(* CODESYS project Parostol_V4.2.project
   CompiledLibraryCompatibilityVersion: CODESYS V3.5 SP16 Patch 3

Project tree, tasks and I/O mapping:
  Device : PLC210, Production association OWEN, order no. 1, version 3.5.17.31
    application Application
      libraries: Standard, * (System); VisuDialogs, * (System); BASIC, 3.3.3.0 (OSCAT); Local Time Library, 3.5.3.50 (Andrew Sorokin); BUILDING, 1.0.0.0 (OSCAT); CmpOwenPidRegs, 3.5.14.33 (Production association OWEN); VisuElemsDateTime Interfaces, * (Intern); CmpBitmapPool, * (System); VisuElemXYChart, 4.1.0.0 (System); CAA DTUtil Extern, 3.5.17.0 (CAA Technical Workgroup); EtherCATStack, 4.2.0.0 (3S - Smart Software Solutions GmbH); Trace Mgr Utils, 4.1.0.0 (Intern); VisuFPlot, 4.1.0.0 (Intern); CmpTargetVisu, 3.5.17.0 (System); CAA Mathematics, 3.5.17.0 (CAA Technical Workgroup); OwenArchiverErrors, 3.5.4.3 (Production association OWEN); Standard64, * (System); OwenStringUtils, 3.5.4.8 (Production association OWEN); cmpSysExec, 3.5.11.30 (OWEN); StringUtils, 3.5.17.0 (System); Util, * (System); Mx210 Assistant, 3.5.11.5 (Production association OWEN)
      Parostol_Zadanie/
        task MainTask (cyclic, interval 20 ms, priority 1) calls PLC_PRG_Stol_1, PLC_PRG_Stol_2, PLC_PRG_Stol_3, PLC_PRG_Stol_4, PLC_PRG_CFC_Davlenie_Stol_1_2, PLC_PRG_CFC_Davlenie_Stol_3_4, PLC_PRG_CFC_Temperatura_Stol_1, PLC_PRG_CFC_Temperatura_Stol_3, PLC_PRG_CFC_Temperatura_Stol_4, PLC_PRG_archive, Connection
        task TrendRecordingTask (cyclic, interval 5000 ms, priority 31) calls VisuTrendStorageAccess.GlobalInstances.g_TrendRecordingManager.CyclicCall
        task VISU_TASK (cyclic, interval 40 ms, priority 0) calls VisuElems.Visu_Prg
        task OwenCloudTask (cyclic, interval 50 ms, priority 31) calls OwenStorage.CLOUD_PRG
        task DatasourcesTask (cyclic, interval 50 ms, priority 31) calls nothing
        task OwenArchiver (cyclic, interval T#100ms, priority 10) calls OwenArchiverDrivers.Archive_Prg
        program PLC_PRG_Stol_1 [CFC]
        function block GRAPH [ST]
        visualisation Zadanie_1
        visualisation HOME_1
        Trend Recording Manager
          Visualization_Trend_Stol_1
          Visualization_Trend_Stol_2
          TrendRecording_CFC_Davlenie_1_2
          TrendRecording_CFC_Temperatura_1
          Visualization_Trend_Stol_3
          Visualization_Trend_Stol_4
        visualisation Visualization_CFC_Davlenie_1_2
        visualisation HOME
        visualisation MnemoScheme
        visualisation Journal
        visualisation Zadanie_2
        program PLC_PRG_Stol_2 [CFC]
        visualisation Visualization_CFC_Temperatura_1
        program PLC_PRG_Stol_3 [CFC]
        program PLC_PRG_Stol_4 [CFC]
        visualisation Zadanie_3
        visualisation Zadanie_4
        visualisation Visualization_CFC_Temperatura_4
        visualisation Visualization_CFC_Temperatura_2
        visualisation Visualization_CFC_Temperatura_3
        visualisation Visualization_CFC_Davlenie_3_4
      CFC_Davlenie_PID/
        program PLC_PRG_CFC_Davlenie_Stol_1_2 [CFC]
        program PLC_PRG_CFC_Davlenie_Stol_3_4 [CFC]
      global variables GVL
      CFC_Temperatura_PID/
        function CheckPidParams_CFC [CFC]
        program PLC_PRG_CFC_Temperatura_Stol_1 [CFC]
        program PLC_PRG_CFC_Temperatura_Stol_4 [CFC]
        program PLC_PRG_CFC_Temperatura_Stol_3 [CFC]
        program PLC_PRG_CFC_Temperatura_Stol_2 [CFC]
      TargetVariables/
        global variables TargetVars
        data type TRG_LeftSide
        data type TRG_Debug
        data type TRG_Drives
        data type TRG_Info
        data type TRG_PLC210
        data type TRG_RTC
        data type TRG_Watchdog
        data type TRG_RightSide
        data type TRG_Buzzer
      global variables PID_GLOBALS
      Списки текстов/
        text list ANR_MODE
        text list ANR_WAVE_COUNT
        text list ERROR_PID
        text list STATE_PID
      archive/
        program PLC_PRG_archive [ST]: act01_DriveInfo
        data type DriveInfo
        function REAL_TO_FWSTRING [ST]
        function BYTE_SIZE_TO_WSTRING [ST]
      program Connection [ST]
      Symbols
      instructions/
        visualisation HELP
        visualisation zapros
        visualisation instrykcai_avtoriz
      global variables NVI_RETAIN
    Ethernet : Ethernet, 3S - Smart Software Solutions GmbH, version 3.5.17.0
        settings: IPAddress = [192,168,0,228]; SubnetMask = [255,255,255,0]; GatewayAddress = [0,0,0,0]; SaveCommunicationSettings = FALSE
      Modbus_TCP_Master : Modbus TCP Master, 3S - Smart Software Solutions GmbH, version 3.5.17.0
        MK210_311_Stol_1_2 : MK210-311, Production association OWEN, version 3.5.11.7
            settings: IPAddress = [192, 168, 0, 230]
            output Application.PLC_PRG_CFC_Davlenie_Stol_1_2.xMore : BOOL  // Битовая маска выходов (запись).Выход 1
            output Application.PLC_PRG_CFC_Davlenie_Stol_1_2.xLess : BOOL  // Битовая маска выходов (запись).Выход 2
            output Application.PLC_PRG_CFC_Temperatura_Stol_1.xLess : BOOL  // Битовая маска выходов (запись).Выход 3
            output Application.PLC_PRG_CFC_Temperatura_Stol_1.xMore : BOOL  // Битовая маска выходов (запись).Выход 4
            unmapped channels: Tmp, Исключить модуль из опроса, Флаг ошибки, Битовая маска входов, Битовая маска выходов (чтение), Битовая маска выходов (запись), Битовая маска диагностики выходов, Значение счетчика, Значение счетчика, Значение счетчика, Значение счетчика, Значение счетчика, Значение счетчика, Сбросить счетчик, Сбросить счетчик, Сбросить счетчик, Сбросить счетчик, Сбросить счетчик, Сбросить счетчик, Период ШИМ (чтение), Период ШИМ (чтение), Период ШИМ (чтение), Период ШИМ (чтение), Период ШИМ (чтение), Период ШИМ (чтение), Период ШИМ (чтение), Период ШИМ (чтение), Период ШИМ (запись), Период ШИМ (запись), Период ШИМ (запись), Период ШИМ (запись), Период ШИМ (запись), Период ШИМ (запись), Период ШИМ (запись), Период ШИМ (запись), Коэффициент заполнения ШИМ (чтение), Коэффициент заполнения ШИМ (чтение), Коэффициент заполнения ШИМ (чтение), Коэффициент заполнения ШИМ (чтение), Коэффициент заполнения ШИМ (чтение),
              Коэффициент заполнения ШИМ (чтение), Коэффициент заполнения ШИМ (чтение), Коэффициент заполнения ШИМ (чтение), Коэффициент заполнения ШИМ (запись), Коэффициент заполнения ШИМ (запись), Коэффициент заполнения ШИМ (запись), Коэффициент заполнения ШИМ (запись), Коэффициент заполнения ШИМ (запись), Коэффициент заполнения ШИМ (запись), Коэффициент заполнения ШИМ (запись), Коэффициент заполнения ШИМ (запись)
        MV210_212_Stol_1_2 : MV210-212, Production association OWEN, version 3.5.11.7
            settings: IPAddress = [192, 168, 0, 231]
            unmapped channels: Tmp, Исключить модуль из опроса, Флаг ошибки, Битовая маска входов, Значение, Значение, Значение, Значение, Значение, Значение, Значение, Значение, Значение счетчика, Значение счетчика, Значение счетчика, Значение счетчика, Значение счетчика, Значение счетчика, Значение счетчика, Значение счетчика, Значение счетчика, Значение счетчика, Значение счетчика, Значение счетчика, Значение счетчика, Значение счетчика, Значение счетчика, Значение счетчика, Значение счетчика, Значение счетчика, Значение счетчика, Значение счетчика, Значение счетчика, Значение счетчика, Значение счетчика, Значение счетчика, Сбросить значение, Сбросить значение, Сбросить значение, Сбросить значение,
              Сбросить значение, Сбросить значение, Сбросить значение, Сбросить значение, Сбросить счетчик, Сбросить счетчик, Сбросить счетчик, Сбросить счетчик, Сбросить счетчик, Сбросить счетчик, Сбросить счетчик, Сбросить счетчик, Сбросить счетчик, Сбросить счетчик, Сбросить счетчик, Сбросить счетчик, Сбросить счетчик, Сбросить счетчик, Сбросить счетчик, Сбросить счетчик, Сбросить счетчик, Сбросить счетчик, Сбросить счетчик, Сбросить счетчик, Сбросить счетчик, Сбросить счетчик, Сбросить счетчик, Сбросить счетчик
        MV210_101_Stol_1_2 : MV210-101, Production association OWEN, version 3.5.11.7
            settings: IPAddress = [192, 168, 0, 232]; Ииспользовать настройки конфигурации = FALSE
            input  Application.PID_GLOBALS.g_rCurrentValue_Temperatura_Stol_1 : REAL  // Вход 3.Значение
            input  Application.PID_GLOBALS.g_rCurrentValue_Davlenie_Podacha_Stol_1_2 : REAL  // Вход 5.Значение
            input  Application.PID_GLOBALS.g_wSampleTime_Davlenie_Stol_1_2 : UINT  // Вход 5.Циклическое время
            input  Application.PID_GLOBALS.g_rCurrentValue_Davlenie_Obratnaja_Stol_1_2 : REAL  // Вход 6.Значение
            unmapped channels: Tmp, Исключить модуль из опроса, Флаг ошибки, Записать настройки, Прочитать настройки, Вход 1 (чтение), Вход 2 (чтение), Вход 3 (чтение), Вход 4 (чтение), Вход 5 (чтение), Вход 6 (чтение), Вход 7 (чтение), Вход 8 (чтение), Вход 1 (запись), Вход 2 (запись), Вход 3 (запись), Вход 4 (запись), Вход 5 (запись), Вход 6 (запись), Вход 7 (запись), Вход 8 (запись), Вход 1, Вход 2, Вход 3, Вход 4, Вход 5, Вход 6, Вход 7, Вход 8
        MK210_311_Stol_3_4 : MK210-311, Production association OWEN, version 3.5.11.7
            settings: IPAddress = [192, 168, 0, 233]
            output Application.PLC_PRG_CFC_Davlenie_Stol_3_4.xMore : BOOL  // Битовая маска выходов (запись).Выход 1
            output Application.PLC_PRG_CFC_Davlenie_Stol_3_4.xLess : BOOL  // Битовая маска выходов (запись).Выход 2
            output Application.PLC_PRG_CFC_Temperatura_Stol_3.xMore : BOOL  // Битовая маска выходов (запись).Выход 3
            output Application.PLC_PRG_CFC_Temperatura_Stol_3.xLess : BOOL  // Битовая маска выходов (запись).Выход 4
            output Application.PLC_PRG_CFC_Temperatura_Stol_4.xMore : BOOL  // Битовая маска выходов (запись).Выход 5
            output Application.PLC_PRG_CFC_Temperatura_Stol_4.xLess : BOOL  // Битовая маска выходов (запись).Выход 6
            unmapped channels: Tmp, Исключить модуль из опроса, Флаг ошибки, Битовая маска входов, Битовая маска выходов (чтение), Битовая маска выходов (запись), Битовая маска диагностики выходов, Значение счетчика, Значение счетчика, Значение счетчика, Значение счетчика, Значение счетчика, Значение счетчика, Сбросить счетчик, Сбросить счетчик, Сбросить счетчик, Сбросить счетчик, Сбросить счетчик, Сбросить счетчик, Период ШИМ (чтение), Период ШИМ (чтение), Период ШИМ (чтение), Период ШИМ (чтение), Период ШИМ (чтение), Период ШИМ (чтение), Период ШИМ (чтение), Период ШИМ (чтение), Период ШИМ (запись), Период ШИМ (запись), Период ШИМ (запись), Период ШИМ (запись), Период ШИМ (запись), Период ШИМ (запись), Период ШИМ (запись), Период ШИМ (запись), Коэффициент заполнения ШИМ (чтение), Коэффициент заполнения ШИМ (чтение), Коэффициент заполнения ШИМ (чтение), Коэффициент заполнения ШИМ (чтение), Коэффициент заполнения ШИМ (чтение),
              Коэффициент заполнения ШИМ (чтение), Коэффициент заполнения ШИМ (чтение), Коэффициент заполнения ШИМ (чтение), Коэффициент заполнения ШИМ (запись), Коэффициент заполнения ШИМ (запись), Коэффициент заполнения ШИМ (запись), Коэффициент заполнения ШИМ (запись), Коэффициент заполнения ШИМ (запись), Коэффициент заполнения ШИМ (запись), Коэффициент заполнения ШИМ (запись), Коэффициент заполнения ШИМ (запись)
        MV210_212_Stol_3_4 : MV210-212, Production association OWEN, version 3.5.11.7
            settings: IPAddress = [192, 168, 0, 234]
            unmapped channels: Tmp, Исключить модуль из опроса, Флаг ошибки, Битовая маска входов, Значение, Значение, Значение, Значение, Значение, Значение, Значение, Значение, Значение счетчика, Значение счетчика, Значение счетчика, Значение счетчика, Значение счетчика, Значение счетчика, Значение счетчика, Значение счетчика, Значение счетчика, Значение счетчика, Значение счетчика, Значение счетчика, Значение счетчика, Значение счетчика, Значение счетчика, Значение счетчика, Значение счетчика, Значение счетчика, Значение счетчика, Значение счетчика, Значение счетчика, Значение счетчика, Значение счетчика, Значение счетчика, Сбросить значение, Сбросить значение, Сбросить значение, Сбросить значение,
              Сбросить значение, Сбросить значение, Сбросить значение, Сбросить значение, Сбросить счетчик, Сбросить счетчик, Сбросить счетчик, Сбросить счетчик, Сбросить счетчик, Сбросить счетчик, Сбросить счетчик, Сбросить счетчик, Сбросить счетчик, Сбросить счетчик, Сбросить счетчик, Сбросить счетчик, Сбросить счетчик, Сбросить счетчик, Сбросить счетчик, Сбросить счетчик, Сбросить счетчик, Сбросить счетчик, Сбросить счетчик, Сбросить счетчик, Сбросить счетчик, Сбросить счетчик, Сбросить счетчик, Сбросить счетчик
        MV210_101_Stol_3_4 : MV210-101, Production association OWEN, version 3.5.11.7
            settings: IPAddress = [192, 168, 0, 235]; Ииспользовать настройки конфигурации = FALSE
            input  Application.PID_GLOBALS.g_rCurrentValue_Temperatura_Stol_3 : REAL  // Вход 1.Значение
            input  Application.PID_GLOBALS.g_rCurrentValue_Temperatura_Stol_4 : REAL  // Вход 3.Значение
            input  Application.PID_GLOBALS.g_rCurrentValue_Davlenie_Podacha_Stol_3_4 : REAL  // Вход 5.Значение
            input  Application.PID_GLOBALS.g_wSampleTime_Davlenie_Stol_3_4 : UINT  // Вход 5.Циклическое время
            input  Application.PID_GLOBALS.g_rCurrentValue_Davlenie_Obratnaja_Stol_3_4 : REAL  // Вход 6.Значение
            unmapped channels: Tmp, Исключить модуль из опроса, Флаг ошибки, Записать настройки, Прочитать настройки, Вход 1 (чтение), Вход 2 (чтение), Вход 3 (чтение), Вход 4 (чтение), Вход 5 (чтение), Вход 6 (чтение), Вход 7 (чтение), Вход 8 (чтение), Вход 1 (запись), Вход 2 (запись), Вход 3 (запись), Вход 4 (запись), Вход 5 (запись), Вход 6 (запись), Вход 7 (запись), Вход 8 (запись), Вход 1, Вход 2, Вход 3, Вход 4, Вход 5, Вход 6, Вход 7, Вход 8
    PLC210_01 : PLC210-02, Production association OWEN, version 3.5.17.3001
        unmapped channels: Канал питания 1, Канал питания 2, Сервисная кнопка, Температура CPU, Переключатель Старт\Стоп
      LeftSide : LeftSide-01, Production association OWEN, version 3.5.17.3001
          unmapped channels: Битовая маска входов, Значение счетчика, Значение счетчика, Значение счетчика, Значение счетчика, Значение счетчика, Значение счетчика, Значение счетчика, Значение счетчика, Значение счетчика, Значение счетчика, Значение счетчика, Значение счетчика, Период импульса, Период импульса, Период импульса, Период импульса, Период импульса, Период импульса, Период импульса, Период импульса, Период импульса, Период импульса, Период импульса, Период импульса, Длительность импульса, Длительность импульса, Длительность импульса, Длительность импульса, Длительность импульса, Длительность импульса, Длительность импульса, Длительность импульса, Длительность импульса, Длительность импульса, Длительность импульса, Длительность импульса, Осталось сгенерировать импульсов, Осталось сгенерировать импульсов, Осталось сгенерировать импульсов,
            Осталось сгенерировать импульсов, Битовая маска диагностики выходов, Счётчик ошибок выхода 1, Счётчик ошибок выхода 2, Счётчик ошибок выхода 3, Счётчик ошибок выхода 4, Количество импульсов AB энкодера 1, Количество импульсов AB энкодера 2, Количество импульсов AB энкодера 3, Количество импульсов AB энкодера 4, Количество импульсов AB энкодера 5, Количество импульсов AB энкодера 6, Количество импульсов ABZ энкодера 1, Количество импульсов ABZ энкодера 2, Количество импульсов ABZ энкодера 3, Количество оборотов ABZ энкодера 1, Количество оборотов ABZ энкодера 2, Количество оборотов ABZ энкодера 3, Битовая маска выходов (запись), Количество импульсов генератора (запись), Количество импульсов генератора (запись), Количество импульсов генератора (запись), Количество импульсов генератора (запись), Выход 1, Выход 2, Выход 3, Выход 4
      RightSide : RightSide-02, Production association OWEN, version 3.5.17.3001
          unmapped channels: Наличие связи, Счетчик ошибок, Битовая маска входов, Битовая маска выходов (запись)
    OwenRTC : OwenRTC, Production association OWEN, version 3.5.17.3001
        input  Application.GVL.hour AT %IB268 : USINT  // Hour
        input  Application.GVL.minute : USINT  // Minute
        input  Application.GVL.day_of_week : USINT  // Day of Week
        unmapped channels: Year, Month, Day, Second, Week of Year, Format Date, Format Time, UTC Offset, NTP Enabled, NTP Error, System Timer, Date And Time, Operating Time, New Year, New Month, New Day, New Hour, New Minute, New Second, New UTC Offset, Set Settings DT, Enable NTP, Prefer Server
    OwenCloud : OwenCloud, Production association OWEN, version 3.5.17.3001
        unmapped channels: OwenCloud enabled, Folder error, Symbol error, No Symbol Config, Status, Enable OwenCloud
    Buzzer : Buzzer, Production association OWEN, version 3.5.17.3001
        unmapped channels: Buzzer enabled, Enable Buzzer, Sound frequency
    Drives : Drives, Production association OWEN, version 3.5.17.3001
        input  Application.PLC_PRG_archive.stPlcMemory.uleFullSize : ULINT  // FS size
        input  Application.PLC_PRG_archive.stPlcMemory.uleUsedSize : ULINT  // FS used
        input  Application.PLC_PRG_archive.stPlcMemory.uleFreeSize : ULINT  // FS free
        input  Application.PLC_PRG_archive.stUsbMemory.xIsMounted : BIT  // USB Mounted
        input  Application.PLC_PRG_archive.stUsbMemory.xUnmountDone : BIT  // USB Unmount done
        input  Application.PLC_PRG_archive.stUsbMemory.uleFullSize : ULINT  // USB size
        input  Application.PLC_PRG_archive.stUsbMemory.uleUsedSize : ULINT  // USB used
        input  Application.PLC_PRG_archive.stUsbMemory.uleFreeSize : ULINT  // USB free
        output Application.PID_GLOBALS.Start_USB_arv : BIT  // Enable Drives
        output Application.PLC_PRG_archive.stUsbMemory.xUnmount : BIT  // USB Unmount
        unmapped channels: MMC Mounted, MMC Unmount done, MMC size, MMC used, MMC free, FS wear, MMC Unmount
    Debug : Debug, Production association OWEN, version 3.5.17.3001
        unmapped channels: RAM used, RAM free, Open files, Processor usage, Core temp, Enable Debug, Debug pause
    Info : Info, Production association OWEN, version 3.5.17.3001
        unmapped channels: VENDOR, DEVICE, SERIAL, RUNTIME, FIRMWARE, LINUX, TARGET, PROJECT, AUTHOR, VERSION, PROFILE, LASTCHANGES
    Watchdog : Watchdog, Production association OWEN, version 3.5.17.3001
        unmapped channels: Exception Handling, Last Exception Code, Last Exception Description, Last Exception Time, Hardware Watchdog Flag, Power Reboot Count, Watchdog Reboot Count, Exception Reboot Count, Command Reboot Count, Reboot, Reset Counters
    OwenArchiver : OwenArchiver, Production association OWEN, version 3.5.4.9
        settings: Имя архива = 'STOL_1'
        output Application.PID_GLOBALS.xGO : BIT  // Запустить архиватор
        output Application.PID_GLOBALS.zGO : BIT  // Команда записи
        input  Application.PLC_PRG_archive.xArchError_1 : USINT  // Код последней ошибки
        input  Application.PLC_PRG_archive.xArchStatus_1 : BIT  // Архиватор работает
        unmapped channels: Запись лога отладки, Путь архивации, Имя архива, Использование буфера записи, Размер архива
      CSVFormat : CSVFormat, Production association OWEN, version 3.5.4.9
      REAL_Variable : REAL Variable, Production association OWEN, version 3.5.4.9
          settings: Описание переменной = 'Выставленное_давление'
          output Application.PLC_PRG_CFC_Davlenie_Stol_1_2.Davlenie_Stol_1_2_rSetPoint : REAL  // Переменная
      BYTE_Stol_1_MINUTE_PONEDEL : BYTE Variable, Production association OWEN, version 3.5.4.9
          settings: Описание переменной = 'Минуты_понедельник'
          output Application.NVI_RETAIN.minuteMondayStolOne : BYTE  // Переменная
      REAL_Stol_1_Y1 : REAL Variable, Production association OWEN, version 3.5.4.9
          settings: Описание переменной = 'Температура_стола'
          output Application.PLC_PRG_Stol_1.Y1 : REAL  // Переменная
      REAL_Stol_1_Y2 : REAL Variable, Production association OWEN, version 3.5.4.9
          settings: Описание переменной = 'Температура_подъема'
          output Application.PLC_PRG_Stol_1.Y2 : REAL  // Переменная
      REAL_Stol_1_Y3 : REAL Variable, Production association OWEN, version 3.5.4.9
          settings: Описание переменной = 'Температура_выдержки'
          output Application.PLC_PRG_Stol_1.Y3 : REAL  // Переменная
      REAL_Stoll_1_HX2 : REAL Variable, Production association OWEN, version 3.5.4.9
          settings: Описание переменной = 'Время_подъема_часы'
          output Application.PLC_PRG_Stol_1.HX2 : REAL  // Переменная
      REAL_Stol_1_MX2 : REAL Variable, Production association OWEN, version 3.5.4.9
          settings: Описание переменной = 'Время_подъема_минуты'
          output Application.PLC_PRG_Stol_1.MX2 : REAL  // Переменная
      REAL_Stol_1_HX3 : REAL Variable, Production association OWEN, version 3.5.4.9
          settings: Описание переменной = 'Время_выдержки_часы'
          output Application.PLC_PRG_Stol_1.HX3 : REAL  // Переменная
      REAL_Stol_1_MX3 : REAL Variable, Production association OWEN, version 3.5.4.9
          settings: Описание переменной = 'Время_выдержки_минуты'
          output Application.PLC_PRG_Stol_1.MX3 : REAL  // Переменная
      BYTE_Stol_1_HOUR_PONEDEL : BYTE Variable, Production association OWEN, version 3.5.4.9
          settings: Описание переменной = 'Час_понедельник'
          output Application.NVI_RETAIN.hourMondayStolOne : BYTE  // Переменная
      BYTE_Stol_1_HOUR_VTORN : BYTE Variable, Production association OWEN, version 3.5.4.9
          settings: Описание переменной = 'Час_вторник'
          output Application.NVI_RETAIN.hourTuesdayStolOne : BYTE  // Переменная
      BYTE_Stol_1_MINUTE_VTORN : BYTE Variable, Production association OWEN, version 3.5.4.9
          settings: Описание переменной = 'Минуты_вторник'
          output Application.NVI_RETAIN.minuteTuesdayStolOne : BYTE  // Переменная
      BYTE_Stol_1_HOUR_SREDA : BYTE Variable, Production association OWEN, version 3.5.4.9
          settings: Описание переменной = 'Час_среды'
          output Application.NVI_RETAIN.hourWednesdayStolOne : BYTE  // Переменная
      BYTE_Stol_1_MINUTE_SREDA : BYTE Variable, Production association OWEN, version 3.5.4.9
          settings: Описание переменной = 'Минуты_среды'
          output Application.NVI_RETAIN.minuteWednesdayStolOne : BYTE  // Переменная
      BYTE_Stol_1_PONEDEL_BYTE : BYTE Variable, Production association OWEN, version 3.5.4.9
          settings: Описание переменной = 'Флаг_понедельника'
          output Application.PLC_PRG_Stol_1.PONEDEL_BYTE : BYTE  // Переменная
      BYTE_Stol_1_VTORN_BYTE : BYTE Variable, Production association OWEN, version 3.5.4.9
          settings: Описание переменной = 'Флаг_вторника'
          output Application.PLC_PRG_Stol_1.VTORN_BYTE : BYTE  // Переменная
      BYTE_Stol_1_SREDA_BYTE : BYTE Variable, Production association OWEN, version 3.5.4.9
          settings: Описание переменной = 'Флаг_среды'
          output Application.PLC_PRG_Stol_1.SREDA_BYTE : BYTE  // Переменная
      BYTE_Stol_1_CHETV_BYTE : BYTE Variable, Production association OWEN, version 3.5.4.9
          settings: Описание переменной = 'Флаг_четверг'
          output Application.PLC_PRG_Stol_1.CHETV_BYTE : BYTE  // Переменная
      BYTE_Stol_1_HOUR_CHETV : BYTE Variable, Production association OWEN, version 3.5.4.9
          settings: Описание переменной = 'Часы_четверг'
          output Application.NVI_RETAIN.hourThursdayStolOne : BYTE  // Переменная
      BYTE_Stol_1_MINUTE_CHETV : BYTE Variable, Production association OWEN, version 3.5.4.9
          settings: Описание переменной = 'Минуты_четверг'
          output Application.NVI_RETAIN.minuteThursdayStolOne : BYTE  // Переменная
      BYTE_Stol_1_PJATN_BYTE : BYTE Variable, Production association OWEN, version 3.5.4.9
          settings: Описание переменной = 'Флаг_пятница'
          output Application.PLC_PRG_Stol_1.PJATN_BYTE : BYTE  // Переменная
      BYTE_Stol_1_HOUR_PJATN : BYTE Variable, Production association OWEN, version 3.5.4.9
          settings: Описание переменной = 'Часы_пятница'
          output Application.NVI_RETAIN.hourFridayStolOne : BYTE  // Переменная
      BYTE_Stol_1_MINUTE_PJATN : BYTE Variable, Production association OWEN, version 3.5.4.9
          settings: Описание переменной = 'Минуты_пятница'
          output Application.NVI_RETAIN.minuteFridayStolOne : BYTE  // Переменная
      BYTE_Stol_1_SUBB_BYTE : BYTE Variable, Production association OWEN, version 3.5.4.9
          settings: Описание переменной = 'Флаг_суббота'
          output Application.PLC_PRG_Stol_1.SUBB_BYTE : BYTE  // Переменная
      BYTE_Stol_1_HOUR_SUBB : BYTE Variable, Production association OWEN, version 3.5.4.9
          settings: Описание переменной = 'Часы_субботы'
          output Application.NVI_RETAIN.hourSaturdayStolOne : BYTE  // Переменная
      BYTE_Stol_1_MINUTE_SUBB : BYTE Variable, Production association OWEN, version 3.5.4.9
          settings: Описание переменной = 'Минуты_субботы'
          output Application.NVI_RETAIN.minuteSaturdayStolOne : BYTE  // Переменная
      BYTE_Stol_1_VOSKR_BYTE : BYTE Variable, Production association OWEN, version 3.5.4.9
          settings: Описание переменной = 'Флаг_воскресенья'
          output Application.PLC_PRG_Stol_1.VOSKR_BYTE : BYTE  // Переменная
      BYTE_Stol_1_HOUR_VOSKR : BYTE Variable, Production association OWEN, version 3.5.4.9
          settings: Описание переменной = 'Часы_воскресенья'
          output Application.NVI_RETAIN.hourSundayStolOne : BYTE  // Переменная
      BYTE_Stol_1_MINUTE_VOSKR : BYTE Variable, Production association OWEN, version 3.5.4.9
          settings: Описание переменной = 'Минуты_воскресенья'
          output Application.NVI_RETAIN.minuteSundayStolOne : BYTE  // Переменная
      BYTE_Stol_1_ACTIVATOR_TIMER_BYTE : BYTE Variable, Production association OWEN, version 3.5.4.9
          settings: Описание переменной = 'Флаг_активации_таймера'
          output Application.PLC_PRG_Stol_1.ACTIVATOR_TIMER_BYTE : BYTE  // Переменная
      REAL_Stol_1_g_rCurrentValue_Temperatura : REAL Variable, Production association OWEN, version 3.5.4.9
          settings: Описание переменной = 'Текущение_значение_температуры'
          output Application.PID_GLOBALS.g_rCurrentValue_Temperatura_Stol_1 : REAL  // Переменная
      REAL_Stol_1_rCurrentValue : REAL Variable, Production association OWEN, version 3.5.4.9
          settings: Описание переменной = 'Показания_давления'
          output Application.PLC_PRG_CFC_Davlenie_Stol_1_2.rCurrentValue : REAL  // Переменная
      STRING_Stol_1_Name : STRING Variable, Production association OWEN, version 3.5.4.9
          settings: Описание переменной = 'Человек_внес_изменения'
          output Application.PLC_PRG_archive.Name : localTypes:STRING  // Переменная
    OwenArchiver_Stol_3_4 : OwenArchiver, Production association OWEN, version 3.5.4.9
        settings: Имя архива = 'STOL_3_4'
        output Application.PID_GLOBALS.xGO : BIT  // Запустить архиватор
        output Application.PID_GLOBALS.yGO : BIT  // Команда записи
        input  Application.PLC_PRG_archive.xArchError_3_4 : USINT  // Код последней ошибки
        input  Application.PLC_PRG_archive.xArchStatus_3_4 : BIT  // Архиватор работает
        unmapped channels: Запись лога отладки, Путь архивации, Имя архива, Использование буфера записи, Размер архива
      CSVFormat_1 : CSVFormat, Production association OWEN, version 3.5.4.9
      BYTE_Stol_3_ACTIVATOR_TIMER_BYTE : BYTE Variable, Production association OWEN, version 3.5.4.9
          settings: Описание переменной = 'Флаг_активации_таймера'
          output Application.PLC_PRG_Stol_3.ACTIVATOR_TIMER_BYTE : BYTE  // Переменная
      BYTE_Stol_3_PONEDEL_BYTE : BYTE Variable, Production association OWEN, version 3.5.4.9
          settings: Описание переменной = 'Флаг_понедельник'
          output Application.PLC_PRG_Stol_3.PONEDEL_BYTE : BYTE  // Переменная
      BYTE_Stol_3_HOUR_PONEDEL : BYTE Variable, Production association OWEN, version 3.5.4.9
          settings: Описание переменной = 'Часы_понедельник'
          output Application.NVI_RETAIN.hourMondayStolThree : BYTE  // Переменная
      BYTE_Stol_3_MINUTE_PONEDEL : BYTE Variable, Production association OWEN, version 3.5.4.9
          settings: Описание переменной = 'Минуты_понедельник'
          output Application.NVI_RETAIN.minuteMondayStolThree : BYTE  // Переменная
      BYTE_Stol_3_VTORN_BYTE : BYTE Variable, Production association OWEN, version 3.5.4.9
          settings: Описание переменной = 'Флаг_вторник'
          output Application.PLC_PRG_Stol_3.VTORN_BYTE : BYTE  // Переменная
      BYTE_Stol_3_HOUR_VTORN : BYTE Variable, Production association OWEN, version 3.5.4.9
          settings: Описание переменной = 'Часы_вторник'
          output Application.NVI_RETAIN.hourTuesdayStolThree : BYTE  // Переменная
      BYTE_Stol_3_MINUTE_VTORN : BYTE Variable, Production association OWEN, version 3.5.4.9
          settings: Описание переменной = 'Минуты_вторник'
          output Application.NVI_RETAIN.minuteTuesdayStolThree : BYTE  // Переменная
      BYTE_Stol_3_SREDA_BYTE : BYTE Variable, Production association OWEN, version 3.5.4.9
          settings: Описание переменной = 'Флаг_среды'
          output Application.PLC_PRG_Stol_3.SREDA_BYTE : BYTE  // Переменная
      BYTE_Stol_3_HOUR_SREDA : BYTE Variable, Production association OWEN, version 3.5.4.9
          settings: Описание переменной = 'Часы_среды'
          output Application.NVI_RETAIN.hourWednesdayStolThree : BYTE  // Переменная
      BYTE_Stol_3_MINUTE_SREDA : BYTE Variable, Production association OWEN, version 3.5.4.9
          settings: Описание переменной = 'Минуты_среды'
          output Application.NVI_RETAIN.minuteWednesdayStolThree : BYTE  // Переменная
      BYTE_Stol_3_CHETV_BYTE : BYTE Variable, Production association OWEN, version 3.5.4.9
          settings: Описание переменной = 'Флаг_четверг'
          output Application.PLC_PRG_Stol_3.CHETV_BYTE : BYTE  // Переменная
      BYTE_Stol_3_HOUR_CHETV : BYTE Variable, Production association OWEN, version 3.5.4.9
          settings: Описание переменной = 'Часы_четверг'
          output Application.NVI_RETAIN.hourThursdayStolThree : BYTE  // Переменная
      BYTE_Stol_3_MINUTE_CHETV : BYTE Variable, Production association OWEN, version 3.5.4.9
          settings: Описание переменной = 'Минуты_четверг'
          output Application.NVI_RETAIN.minuteThursdayStolThree : BYTE  // Переменная
      BYTE_Stol_3_PJATN_BYTE : BYTE Variable, Production association OWEN, version 3.5.4.9
          settings: Описание переменной = 'Флаг_пятница'
          output Application.PLC_PRG_Stol_3.PJATN_BYTE : BYTE  // Переменная
      BYTE_Stol_3_HOUR_PJATN : BYTE Variable, Production association OWEN, version 3.5.4.9
          settings: Описание переменной = 'Часы_пятницы'
          output Application.NVI_RETAIN.hourFridayStolThree : BYTE  // Переменная
      BYTE_Stol_3_MINUTE_PJATN : BYTE Variable, Production association OWEN, version 3.5.4.9
          settings: Описание переменной = 'Минуты_пятницы'
          output Application.NVI_RETAIN.minuteFridayStolThree : BYTE  // Переменная
      BYTE_Stol_3_SUBB_BYTE : BYTE Variable, Production association OWEN, version 3.5.4.9
          settings: Описание переменной = 'Флаг_субботы'
          output Application.PLC_PRG_Stol_3.SUBB_BYTE : BYTE  // Переменная
      BYTE_Stol_3_HOUR_SUBB : BYTE Variable, Production association OWEN, version 3.5.4.9
          settings: Описание переменной = 'Часы_субботы'
          output Application.NVI_RETAIN.hourSaturdayStolThree : BYTE  // Переменная
      BYTE_Stol_3_MINUTE_SUBB : BYTE Variable, Production association OWEN, version 3.5.4.9
          settings: Описание переменной = 'Минуты_субботы'
          output Application.NVI_RETAIN.minuteSaturdayStolThree : BYTE  // Переменная
      BYTE_Stol_3_VOSKR_BYTE : BYTE Variable, Production association OWEN, version 3.5.4.9
          settings: Описание переменной = 'Флаг_воскресенья'
          output Application.PLC_PRG_Stol_3.VOSKR_BYTE : BYTE  // Переменная
      BYTE_Stol_3_HOUR_VOSKR : BYTE Variable, Production association OWEN, version 3.5.4.9
          settings: Описание переменной = 'Часы_воскресенья'
          output Application.NVI_RETAIN.hourSundayStolThree : BYTE  // Переменная
      BYTE_Stol_3_MINUTE_VOSKR : BYTE Variable, Production association OWEN, version 3.5.4.9
          settings: Описание переменной = 'Минуты_воскресенья'
          output Application.NVI_RETAIN.minuteSundayStolThree : BYTE  // Переменная
      REAL_Stol_3_Y1 : REAL Variable, Production association OWEN, version 3.5.4.9
          settings: Описание переменной = 'Температура_стола'
          output Application.PLC_PRG_Stol_3.Y1 : REAL  // Переменная
      REAL_Stol_3_Y2 : REAL Variable, Production association OWEN, version 3.5.4.9
          settings: Описание переменной = 'Температура_подъёма'
          output Application.PLC_PRG_Stol_3.Y2 : REAL  // Переменная
      REAL_Stol_3_Y3 : REAL Variable, Production association OWEN, version 3.5.4.9
          settings: Описание переменной = 'Температура_выдержки'
          output Application.PLC_PRG_Stol_3.Y3 : REAL  // Переменная
      REAL_Stol_3_HX2 : REAL Variable, Production association OWEN, version 3.5.4.9
          settings: Описание переменной = 'Часы_подъёма'
          output Application.PLC_PRG_Stol_3.HX2 : REAL  // Переменная
      REAL_Stol_3_MX2 : REAL Variable, Production association OWEN, version 3.5.4.9
          settings: Описание переменной = 'Минуты_подъёма'
          output Application.PLC_PRG_Stol_3.MX2 : REAL  // Переменная
      REAL_Stol_3_HX3 : REAL Variable, Production association OWEN, version 3.5.4.9
          settings: Описание переменной = 'Часы_выдержки'
          output Application.PLC_PRG_Stol_3.HX3 : REAL  // Переменная
      REAL_Stol_3_MX3 : REAL Variable, Production association OWEN, version 3.5.4.9
          settings: Описание переменной = 'Минуты_выдержки'
          output Application.PLC_PRG_Stol_3.MX3 : REAL  // Переменная
      REAL_Davlenie_Stol_3_4_rSetPoint : REAL Variable, Production association OWEN, version 3.5.4.9
          settings: Описание переменной = 'Выставленное_давление'
          output Application.PLC_PRG_CFC_Davlenie_Stol_3_4.Davlenie_Stol_3_4_rSetPoint : REAL  // Переменная
      BYTE_Stol_4_ACTIVATOR_TIMER_BYTE : BYTE Variable, Production association OWEN, version 3.5.4.9
          settings: Описание переменной = 'Флаг_активации_таймера'
          output Application.PLC_PRG_Stol_4.ACTIVATOR_TIMER_BYTE : BYTE  // Переменная
      BYTE_Stol_4_PONEDEL_BYTE : BYTE Variable, Production association OWEN, version 3.5.4.9
          settings: Описание переменной = 'Флаг_понедельника'
          output Application.PLC_PRG_Stol_4.PONEDEL_BYTE : BYTE  // Переменная
      BYTE_Stol_4_HOUR_PONEDEL : BYTE Variable, Production association OWEN, version 3.5.4.9
          settings: Описание переменной = 'Часы_понедельника'
          output Application.NVI_RETAIN.hourMondayStolFour : BYTE  // Переменная
      BYTE_Stol_4_MINUTE_PONEDEL : BYTE Variable, Production association OWEN, version 3.5.4.9
          settings: Описание переменной = 'Минуты_понедельника'
          output Application.NVI_RETAIN.minuteMondayStolFour : BYTE  // Переменная
      BYTE_Stol_4_VTORN_BYTE : BYTE Variable, Production association OWEN, version 3.5.4.9
          settings: Описание переменной = 'Флаг_вторник'
          output Application.PLC_PRG_Stol_4.VTORN_BYTE : BYTE  // Переменная
      BYTE_Stol_4_HOUR_VTORN : BYTE Variable, Production association OWEN, version 3.5.4.9
          settings: Описание переменной = 'Часы_вторника'
          output Application.NVI_RETAIN.hourTuesdayStolFour : BYTE  // Переменная
      BYTE_Stol_4_MINUTE_VTORN : BYTE Variable, Production association OWEN, version 3.5.4.9
          settings: Описание переменной = 'Минуты_вторника'
          output Application.NVI_RETAIN.minuteTuesdayStolFour : BYTE  // Переменная
      BYTE_Stol_4_SREDA_BYTE : BYTE Variable, Production association OWEN, version 3.5.4.9
          settings: Описание переменной = 'Флаг_среды'
          output Application.PLC_PRG_Stol_4.SREDA_BYTE : BYTE  // Переменная
      BYTE_Stol_4_HOUR_SREDA : BYTE Variable, Production association OWEN, version 3.5.4.9
          settings: Описание переменной = 'Часы_среды'
          output Application.NVI_RETAIN.hourWednesdayStolFour : BYTE  // Переменная
      BYTE_Stol_4_MINUTE_SREDA : BYTE Variable, Production association OWEN, version 3.5.4.9
          settings: Описание переменной = 'Минуты_среды'
          output Application.NVI_RETAIN.minuteWednesdayStolFour : BYTE  // Переменная
      BYTE_Stol_4_CHETV_BYTE : BYTE Variable, Production association OWEN, version 3.5.4.9
          settings: Описание переменной = 'Флаг_четверга'
          output Application.PLC_PRG_Stol_4.CHETV_BYTE : BYTE  // Переменная
      BYTE_Stol_4_HOUR_CHETV : BYTE Variable, Production association OWEN, version 3.5.4.9
          settings: Описание переменной = 'Часы_четверга'
          output Application.NVI_RETAIN.hourThursdayStolFour : BYTE  // Переменная
      BYTE_Stol_4_MINUTE_CHETV : BYTE Variable, Production association OWEN, version 3.5.4.9
          settings: Описание переменной = 'Минуты_четверга'
          output Application.NVI_RETAIN.minuteThursdayStolFour : BYTE  // Переменная
      BYTE_Stol_4_PJATN_BYTE : BYTE Variable, Production association OWEN, version 3.5.4.9
          settings: Описание переменной = 'Флаг_пятница'
          output Application.PLC_PRG_Stol_4.PJATN_BYTE : BYTE  // Переменная
      BYTE_Stol_4_HOUR_PJATN : BYTE Variable, Production association OWEN, version 3.5.4.9
          settings: Описание переменной = 'Часы_пятницы'
          output Application.NVI_RETAIN.hourFridayStolFour : BYTE  // Переменная
      BYTE_Stol_4_MINUTE_PJATN : BYTE Variable, Production association OWEN, version 3.5.4.9
          settings: Описание переменной = 'Минуты_пятницы'
          output Application.NVI_RETAIN.minuteFridayStolFour : BYTE  // Переменная
      BYTE_Stol_4_SUBB_BYTE : BYTE Variable, Production association OWEN, version 3.5.4.9
          settings: Описание переменной = 'Флаг_субботы'
          output Application.PLC_PRG_Stol_4.SUBB_BYTE : BYTE  // Переменная
      BYTE_Stol_4_HOUR_SUBB : BYTE Variable, Production association OWEN, version 3.5.4.9
          settings: Описание переменной = 'Часы_субботы'
          output Application.NVI_RETAIN.hourSaturdayStolFour : BYTE  // Переменная
      BYTE_Stol_4_MINUTE_SUBB : BYTE Variable, Production association OWEN, version 3.5.4.9
          settings: Описание переменной = 'Минуты_субботы'
          output Application.NVI_RETAIN.minuteSaturdayStolFour : BYTE  // Переменная
      BYTE_Stol_4_VOSKR_BYTE : BYTE Variable, Production association OWEN, version 3.5.4.9
          settings: Описание переменной = 'Флаг_воскресенья'
          output Application.PLC_PRG_Stol_4.VOSKR_BYTE : BYTE  // Переменная
      BYTE_Stol_4_HOUR_VOSKR : BYTE Variable, Production association OWEN, version 3.5.4.9
          settings: Описание переменной = 'Часы_воскресенья'
          output Application.NVI_RETAIN.hourSundayStolFour : BYTE  // Переменная
      BYTE_Stol_4_MINUTE_VOSKR : BYTE Variable, Production association OWEN, version 3.5.4.9
          settings: Описание переменной = 'Минуты_воскресенья'
          output Application.NVI_RETAIN.minuteSundayStolFour : BYTE  // Переменная
      REAL_Stol_4_Y1 : REAL Variable, Production association OWEN, version 3.5.4.9
          settings: Описание переменной = 'Температура_стола'
          output Application.PLC_PRG_Stol_4.Y1 : REAL  // Переменная
      REAL_Stol_4_Y2 : REAL Variable, Production association OWEN, version 3.5.4.9
          settings: Описание переменной = 'Температура_подъёма'
          output Application.PLC_PRG_Stol_4.Y2 : REAL  // Переменная
      REAL_Stol_4_Y3 : REAL Variable, Production association OWEN, version 3.5.4.9
          settings: Описание переменной = 'Температура_выдержки'
          output Application.PLC_PRG_Stol_4.Y3 : REAL  // Переменная
      REAL_Stol_4_HX2 : REAL Variable, Production association OWEN, version 3.5.4.9
          settings: Описание переменной = 'Часы_подъёма'
          output Application.PLC_PRG_Stol_4.HX2 : REAL  // Переменная
      REAL_Stol_4_MX2 : REAL Variable, Production association OWEN, version 3.5.4.9
          settings: Описание переменной = 'Минуты_подъёма'
          output Application.PLC_PRG_Stol_4.MX2 : REAL  // Переменная
      REAL_Stol_4_HX3 : REAL Variable, Production association OWEN, version 3.5.4.9
          settings: Описание переменной = 'Часы_выдержки'
          output Application.PLC_PRG_Stol_4.HX3 : REAL  // Переменная
      REAL_Stol_4_MX3 : REAL Variable, Production association OWEN, version 3.5.4.9
          settings: Описание переменной = 'Минуты_выдержки'
          output Application.PLC_PRG_Stol_4.MX3 : REAL  // Переменная
      REAL_Stol_3_g_rCurrentValue_Temperatura : REAL Variable, Production association OWEN, version 3.5.4.9
          settings: Описание переменной = 'Текущение_значение_температуры'
          output Application.PID_GLOBALS.g_rCurrentValue_Temperatura_Stol_3 : REAL  // Переменная
      REAL_Stol_3_4_rCurrentValue : REAL Variable, Production association OWEN, version 3.5.4.9
          settings: Описание переменной = 'Показания_давления'
          output Application.PLC_PRG_CFC_Davlenie_Stol_3_4.rCurrentValue : REAL  // Переменная
      REAL_Stol_4_g_rCurrentValue_Temperatura : REAL Variable, Production association OWEN, version 3.5.4.9
          settings: Описание переменной = 'Текущение_значение_температуры'
          output Application.PID_GLOBALS.g_rCurrentValue_Temperatura_Stol_4 : REAL  // Переменная
      STRING_Stol_3_4_Name : STRING Variable, Production association OWEN, version 3.5.4.9
          settings: Описание переменной = 'Человек_внес_изменения'
          output Application.PLC_PRG_archive.Name : localTypes:STRING  // Переменная
  libraries: VisuSymbols, 4.1.0.0 (System)
  text list GlobalTextList
  text list System
  GlobalImagePool
  function block POU_LIN_TRAFO [ST]
  global variables GVL
*)

// Device/Application/TargetVariables/TRG_LeftSide
TYPE TRG_LeftSide :
STRUCT
	xFastDi01:				BOOL;
	xFastDi02:				BOOL;
	xFastDi03:				BOOL;
	xFastDi04:				BOOL;
	xFastDi05:				BOOL;
	xFastDi06:				BOOL;
	xFastDi07:				BOOL;
	xFastDi08:				BOOL;
	xFastDi09: 				BOOL;
	xFastDi10:				BOOL;
	xFastDi11:				BOOL;
	xFastDi12:				BOOL;
	
	xDo01:					BOOL;
	xDo02:					BOOL;
	xDo03:					BOOL;
	xDo04:					BOOL;
	
	udiCounterFastDi01:		UDINT;
	udiCounterFastDi02:		UDINT;
	udiCounterFastDi03:		UDINT;
	udiCounterFastDi04:		UDINT;
	udiCounterFastDi05:		UDINT;
	udiCounterFastDi06:		UDINT;
	udiCounterFastDi07:		UDINT;
	udiCounterFastDi08:		UDINT;
	udiCounterFastDi09:		UDINT;
	udiCounterFastDi10:		UDINT;
	udiCounterFastDi11:		UDINT;
	udiCounterFastDi12:		UDINT;
	
	udiPulseDurationFastDi01:	UDINT;
	udiPulseDurationFastDi02:	UDINT;
	udiPulseDurationFastDi03:	UDINT;
	udiPulseDurationFastDi04:	UDINT;
	udiPulseDurationFastDi05:	UDINT;
	udiPulseDurationFastDi06:	UDINT;
	udiPulseDurationFastDi07:	UDINT;
	udiPulseDurationFastDi08:	UDINT;
	udiPulseDurationFastDi09:	UDINT;
	udiPulseDurationFastDi10:	UDINT;
	udiPulseDurationFastDi11:	UDINT;
	udiPulseDurationFastDi12:	UDINT;

	udiPulsePeriodFastDi01:		UDINT;
	udiPulsePeriodFastDi02:		UDINT;
	udiPulsePeriodFastDi03:		UDINT;
	udiPulsePeriodFastDi04:		UDINT;
	udiPulsePeriodFastDi05:		UDINT;
	udiPulsePeriodFastDi06:		UDINT;
	udiPulsePeriodFastDi07:		UDINT;
	udiPulsePeriodFastDi08:		UDINT;
	udiPulsePeriodFastDi09:		UDINT;
	udiPulsePeriodFastDi10:		UDINT;
	udiPulsePeriodFastDi11:		UDINT;
	udiPulsePeriodFastDi12:		UDINT;
	
	udiGenPulseCountDo01:	    UDINT;
	udiGenPulseCountDo02:	    UDINT;
	udiGenPulseCountDo03:	    UDINT;
	udiGenPulseCountDo04:	    UDINT;
	
	udiGenPulseCountLeftDo01:	UDINT;
	udiGenPulseCountLeftDo02:	UDINT;
	udiGenPulseCountLeftDo03:	UDINT;
	udiGenPulseCountLeftDo04:	UDINT;
	
	udiPwmDutyCycleDo01:		UDINT;
	udiPwmDutyCycleDo02:		UDINT;
	udiPwmDutyCycleDo03:		UDINT;
	udiPwmDutyCycleDo04:		UDINT;
	
	udiPulseCounterAbEncoder01: DINT;
	udiPulseCounterAbEncoder02: DINT;
	udiPulseCounterAbEncoder03: DINT;
	udiPulseCounterAbEncoder04: DINT;
	udiPulseCounterAbEncoder05: DINT;
	udiPulseCounterAbEncoder06: DINT;
	
	udiPulseCounterAbzEncoder01: DINT;
	udiPulseCounterAbzEncoder02: DINT;
	udiPulseCounterAbzEncoder03: DINT;
	
	udiTurnCounterAbzEncoder01: DINT;
	udiTurnCounterAbzEncoder02: DINT;
	udiTurnCounterAbzEncoder03: DINT;
END_STRUCT
END_TYPE

// Device/Application/TargetVariables/TRG_Debug
TYPE TRG_Debug :
STRUCT
	xEnable: 			BOOL;
	udiPollingTime:		UDINT;
	udiRamUsedSize:		UDINT;
	udiRamFreeSize:		UDINT;
	udiCountHandles:	UDINT;
	udiProcUsage:		UDINT;
END_STRUCT
END_TYPE

// Device/Application/TargetVariables/TRG_Drives
TYPE TRG_Drives :
STRUCT
	xEnable:			BOOL;
	
	uliFsFullSize: 		ULINT;
	uliFsUsedSize: 		ULINT;
	uliFsFreeSize: 		ULINT;
	
	xUsbMounted:		BOOL;
	xUsbUnmount:		BOOL;
	xUsbUnmountDone:	BOOL;
	
	uliUsbFullSize: 	ULINT;
	uliUsbUsedSize: 	ULINT;
	uliUsbFreeSize: 	ULINT;
	
	xSdMounted:			BOOL;
	xSdUnmount:			BOOL;
	xSdUnmountDone:		BOOL;
	
	uliSdFullSize: 		ULINT;
	uliSdUsedSize: 		ULINT;
	uliSdFreeSize: 		ULINT;
END_STRUCT
END_TYPE

// Device/Application/TargetVariables/TRG_Info
TYPE TRG_Info :
STRUCT
	sVendorName: 			STRING;
	sDeviceName: 			STRING;
	sSerialId: 				STRING;
	sRuntimeVersion:		STRING;
	sFirmwareVersion: 		STRING;
	sLinuxVersion: 			STRING;
	sNeedTargetVersion:		STRING;
	
	sProjectName:			STRING;
	sAuthorName:			STRING;
	sProjectVersion:		STRING;
	sProjectProfile:		STRING;
	dtProjectLastChanges:	DT;
END_STRUCT
END_TYPE

// Device/Application/TargetVariables/TRG_PLC210
TYPE TRG_PLC210 :
STRUCT
	xPowerInput1:	 BOOL;
	xPowerInput2: 	 BOOL;
	xServiceButton:  BOOL;
	rCpuTemp:		 REAL;
END_STRUCT
END_TYPE

// Device/Application/TargetVariables/TRG_RTC
TYPE TRG_RTC :
STRUCT
	uiGetYear:			UINT;
	usiGetMonth:		USINT;
	usiGetDay:			USINT;
	usiGetHour:			USINT;
	usiGetMinute:		USINT;
	usiGetSecond:		USINT;
	usiGetDayOfWeek:	USINT;
	usiGetWeekOfYear:	USINT;
	sGetFormatDate:		STRING;
	sGetFormatTime:		STRING;
	siGetUtcOffset:		SINT;
	dtDateAndTime:		DT;
	
	
	uiSetYear:			UINT;
	usiSetMonth:		USINT;
	usiSetDay:			USINT;
	usiSetHour:			USINT;
	usiSetMinute:		USINT;
	usiSetSecond:		USINT;
	siSetUtcOffset:		SINT;
	xUpdateSettings:	BOOL;
	
	xEnableNtp:			BOOL;
	xIsNtpEnabled:		BOOL;
	sPreferNtpServer:	STRING;
	usiNtpErrorCode:	USINT;
	
	ltSystemTick:		LTIME;
END_STRUCT
END_TYPE

// Device/Application/TargetVariables/TRG_Watchdog
TYPE TRG_Watchdog :
STRUCT
	//eHandlingType:						Watchdog.ExceptionHandling;
	udiLastExceptionCode:				UDINT;
	sLastExceptionText:					STRING;
	dtLastExceptionTime:				DT;
	xIsHardwareWatchdogReboot:			BOOL;
	xDoReboot:							BOOL;
	usiPowerRebootCount:				USINT;
	usiExceptionRebootCount:			USINT;
	usiCommandRebootCount:				USINT;
	usiHardwareWatchdogRebootCount:		USINT;
	xResetCounters:						BOOL;
END_STRUCT
END_TYPE

// Device/Application/TargetVariables/TRG_RightSide
TYPE TRG_RightSide :
STRUCT
	xSystemBusLink:		BOOL;
	udiSystemBusError:  UDINT;
	
	xDo05:				BOOL;
	xDo06:				BOOL;
	xDo07:				BOOL;
	xDo08:				BOOL;
	xDo09:				BOOL;
	xDo10:				BOOL;
	xDo11:				BOOL;
	xDo12:				BOOL;
	xDo13:				BOOL;
	xDo14:				BOOL;
	xDo15:				BOOL;
	xDo16:				BOOL;
	xDo17:				BOOL;
	xDo18:				BOOL;
END_STRUCT
END_TYPE

// Device/Application/TargetVariables/TRG_Buzzer
TYPE TRG_Buzzer :
STRUCT
	xGet:	BOOL;
	xSet:	BOOL;
END_STRUCT
END_TYPE

// Device/Application/archive/DriveInfo
TYPE DriveInfo :
STRUCT
	xIsMounted:			BOOL;		// флаг "накопитель примонтирован"
	xUnmount:			BOOL;		// сигнал размонтирования накопителя
	xUnmountDone:		BOOL;		// флаг "накопитель размонтирован"
	
	uleFullSize:		ULINT;		// общий объем доступного дискового пространства (в байтах)
	uleUsedSize:		ULINT;		// занятый объем доступного дискового пространства (в байтах)
	uleFreeSize:		ULINT;		// свободный объем доступного дискового пространства (в байтах)
	
	wsFullSize:		WSTRING;		// общий объем доступного дискового пространства (форматированная строка) 
	wsUsedSize:		WSTRING;		// занятый объем доступного дискового пространства (форматированная строка)
	wsFreeSize:		WSTRING;		// свободный объем доступного дискового пространства (форматированная строка)
END_STRUCT
END_TYPE

// GVL
{attribute 'qualified_only'}
VAR_GLOBAL
END_VAR

// Device/Application/GVL
{attribute 'qualified_only'}
VAR_GLOBAL
	hour:USINT;
	minute:USINT;
	day_of_week:USINT;
END_VAR

// Device/Application/TargetVariables/TargetVars
{attribute 'qualified_only'}
VAR_GLOBAL
	stBuzzer:	 	TRG_Buzzer;
	stDebug: 		TRG_Debug;
	stDrives: 		TRG_Drives;
	stRtc:			TRG_RTC;
	stInfo:			TRG_Info;
	stWatchdog:		TRG_Watchdog;
	stPlc210:	 	TRG_PLC210;
	stLeftSide:		TRG_LeftSide;
	stRightSide:	TRG_RightSide;
	
	//stNetwork:	 TRG_Network;
END_VAR

// Device/Application/PID_GLOBALS
{attribute 'qualified_only'}
VAR_GLOBAL
	
 	Temperatura_Stol_1_rSetPoint:			REAL;			// Уставка задания
	Temperatura_Stol_2_rSetPoint:			REAL;			// Уставка задания
	Temperatura_Stol_3_rSetPoint: 			REAL;			// Уставка задания
	Temperatura_Stol_4_rSetPoint: 			REAL;			// Уставка задания
		
	g_rCurrentValue_Temperatura_Stol_1:		REAL;			// Измеренное значение регулируемой величины
	g_rCurrentValue_Temperatura_Stol_2:		REAL;			// Измеренное значение регулируемой величины
	g_rCurrentValue_Temperatura_Stol_3:		REAL;			// Измеренное значение регулируемой величины
	g_rCurrentValue_Temperatura_Stol_4:		REAL;			// Измеренное значение регулируемой величины
		
	g_rCurrentValue_Davlenie_Podacha_Stol_1_2:			REAL;			// Измеренное значение регулируемой величины 
	g_rCurrentValue_Davlenie_Obratnaja_Stol_1_2:		REAL;			// Измеренное значение регулируемой величины
	
	
	g_rCurrentValue_Davlenie_Podacha_Stol_3_4:			REAL;			// Измеренное значение регулируемой величины 
	g_rCurrentValue_Davlenie_Obratnaja_Stol_3_4:		REAL;			// Измеренное значение регулируемой величины
	
	g_wSampleTime_Davlenie_Stol_1_2: 					WORD;			// Циклическое время обновления входа измеренного значение регулируемой величины (в сотых долях секунды)
	g_wSampleTime_Davlenie_Stol_3_4: 					WORD;			// Циклическое время обновления входа измеренного значение регулируемой величины (в сотых долях секунды)
	
	xOut_Less_Davlenie_Stol_1_2:							BOOL;			// Сигнал на закрытие ИМ
	xOut_More_Davlenie_Stol_1_2:							BOOL;			// Сигнал на открытие ИМ
	
	xOut_Less_Davlenie_Stol_3_4:							BOOL;			// Сигнал на закрытие ИМ
	xOut_More_Davlenie_Stol_3_4:							BOOL;			// Сигнал на открытие ИМ
	
	// переменные архиватора
	xGO:										BOOL := TRUE;				// Старт записи в архив
	yGO:										BOOL;						// Команда на записи в архив 3 и 4 стол
	zGO:										BOOL;						// Команда на записи в архив 1 стола
	Start_USB_arv:								BOOL := TRUE;				// Монтирует при запуске USB-накопитель
	
	
END_VAR

// Device/Application/NVI_RETAIN
{attribute 'qualified_only'}
VAR_GLOBAL RETAIN
	dateWeekStolOneTwo:		WORD := 1;	(*	0-й бит - Активировать таймер Стол 1
											1-й бит - Понедельник Стол 1
											2-й бит - Вторник Стол 1
											3-й бит - Среда Стол 1
											4-й бит - Четверг Стол 1
											5-й бит - Пятница Стол 1
											6-й бит - Суббота Стол 1
											7-й бит - Воскресенье Стол 1 *)
	
	hourMondayStolOne:			BYTE;		// Часы запуска первого стола в понедельник			
	hourTuesdayStolOne:			BYTE;		// Часы запуска первого стола во вторник	
	hourWednesdayStolOne:		BYTE;		// Часы запуска первого стола в среда	
	hourThursdayStolOne:		BYTE;		// Часы запуска первого стола в четверг		
	hourFridayStolOne:			BYTE;		// Часы запуска первого стола в пятница	
	hourSaturdayStolOne:		BYTE;		// Часы запуска первого стола в суббота	
	hourSundayStolOne:			BYTE;		// Часы запуска первого стола в воскресенье		

	minuteMondayStolOne:		BYTE;		// Минуты запуска первого стола в понедельник			
	minuteTuesdayStolOne:		BYTE;		// Минуты запуска первого стола во вторник	
	minuteWednesdayStolOne:		BYTE;		// Минуты запуска первого стола в среда	
	minuteThursdayStolOne:		BYTE;		// Минуты запуска первого стола в четверг		
	minuteFridayStolOne:		BYTE;		// Минуты запуска первого стола в пятница	
	minuteSaturdayStolOne:		BYTE;		// Минуты запуска первого стола в суббота	
	minuteSundayStolOne:		BYTE;		// Минуты запуска первого стола в воскресенье						
	
	dateWeekStolThreeFour:	WORD := 257;	(*	0-й бит - Активировать таймер Стол 3
											1-й бит - Понедельник Стол 3
											2-й бит - Вторник Стол 3
											3-й бит - Среда Стол 3
											4-й бит - Четверг Стол 3
											5-й бит - Пятница Стол 3
											6-й бит - Суббота Стол 3
											7-й бит - Воскресенье Стол 3
											8-й бит - Активировать таймер Стол 4
											9-й бит - Понедельник Стол 4
											10-й бит - Вторник Стол 4
											11-й бит - Среда Стол 4
											12-й бит - Четверг Стол 4
											13-й бит - Пятница Стол 4
											14-й бит - Суббота Стол 4
											15-й бит - Воскресенье Стол 4 *)
											
	hourMondayStolThree:		BYTE;		// Часы запуска третьего стола в понедельник			
	hourTuesdayStolThree:		BYTE;		// Часы запуска третьего стола во вторник	
	hourWednesdayStolThree:		BYTE;		// Часы запуска третьего стола в среда	
	hourThursdayStolThree:		BYTE;		// Часы запуска третьего стола в четверг		
	hourFridayStolThree:		BYTE;		// Часы запуска третьего стола в пятница	
	hourSaturdayStolThree:		BYTE;		// Часы запуска третьего стола в суббота	
	hourSundayStolThree:		BYTE;		// Часы запуска третьего стола в воскресенье		

	minuteMondayStolThree:		BYTE;		// Минуты запуска третьего стола в понедельник			
	minuteTuesdayStolThree:		BYTE;		// Минуты запуска третьего стола во вторник	
	minuteWednesdayStolThree:	BYTE;		// Минуты запуска третьего стола в среда	
	minuteThursdayStolThree:	BYTE;		// Минуты запуска третьего стола в четверг		
	minuteFridayStolThree:		BYTE;		// Минуты запуска третьего стола в пятница	
	minuteSaturdayStolThree:	BYTE;		// Минуты запуска третьего стола в суббота	
	minuteSundayStolThree:		BYTE;		// Минуты запуска третьего стола в воскресенье
	
	hourMondayStolFour:			BYTE;		// Часы запуска четвёртого стола в понедельник			
	hourTuesdayStolFour:		BYTE;		// Часы запуска четвёртого стола во вторник	
	hourWednesdayStolFour:		BYTE;		// Часы запуска четвёртого стола в среда	
	hourThursdayStolFour:		BYTE;		// Часы запуска четвёртого стола в четверг		
	hourFridayStolFour:			BYTE;		// Часы запуска четвёртого стола в пятница	
	hourSaturdayStolFour:		BYTE;		// Часы запуска четвёртого стола в суббота	
	hourSundayStolFour:			BYTE;		// Часы запуска четвёртого стола в воскресенье		

	minuteMondayStolFour:		BYTE;		// Минуты запуска четвёртого стола в понедельник			
	minuteTuesdayStolFour:		BYTE;		// Минуты запуска четвёртого стола во вторник	
	minuteWednesdayStolFour:	BYTE;		// Минуты запуска четвёртого стола в среда	
	minuteThursdayStolFour:		BYTE;		// Минуты запуска четвёртого стола в четверг		
	minuteFridayStolFour:		BYTE;		// Минуты запуска четвёртого стола в пятница	
	minuteSaturdayStolFour:		BYTE;		// Минуты запуска четвёртого стола в суббота	
	minuteSundayStolFour:		BYTE;		// Минуты запуска четвёртого стола в воскресенье
END_VAR

// Device/Application/Parostol_Zadanie/PLC_PRG_Stol_1
PROGRAM PLC_PRG_Stol_1
VAR
	
	TON1: 						TON;
	X: 							REAL;
	X1: 						BYTE:=1;

	X2:							REAL;
	X3: 						REAL;
	X4: 						BYTE:=1;
	Y4: 						REAL;
	GR1: 						GRAPH;
	
	arrHist1:					ARRAY [0..3] OF REAL;
	
	
	DHTV:						REAL;
	RESULTAT: 					TIME;
	RES: 						TIME;
	RS_01: 						RS;
	R_TRIG_01: 					R_TRIG;
	INDIKATOR: 					BOOL;
	R_TRIG_02: 					R_TRIG;
	STOP: 						BOOL;
	R_TRIG_03: 					R_TRIG;
	
	// Конвертация для архивации
	ACTIVATOR_TIMER_BYTE:		BYTE;
	PONEDEL_BYTE:				BYTE;					
	VTORN_BYTE:					BYTE;		
	SREDA_BYTE:					BYTE;
	CHETV_BYTE:					BYTE;
	PJATN_BYTE:					BYTE;
	SUBB_BYTE:					BYTE;
	VOSKR_BYTE:					BYTE;
	
	ostanovka: 					BOOL;						// Переменная для команды запуска закрытия 3-х ходового
END_VAR
VAR RETAIN
	
	START: 						BOOL;
	
	Y1:							REAL; 					// Начальная температу
	Y2: 						REAL;					// Температура подъёма
	Y3: 						REAL;					// Температура выдержки
	
	HX2: 						REAL;					// Время подъёма часы
	MX2: 						REAL;					// Время подъёма минуты
	HX3: 						REAL;					// Время выдержки часы
	MX3: 						REAL;					// Время выдержки минуты
END_VAR
VAR // added by the converter: edge detectors and wires of the graphical bodies
    _w1, _w3, _w19, _w20, _w21 : BYTE;
    _w2, _w17, _w23 : REAL;
    _w4, _w6, _w7, _w8, _w9, _w10, _w11, _w12, _w13, _w14, _w15, _w16, _w18 : BOOL;
    _w5, _w22 : ANY;
END_VAR

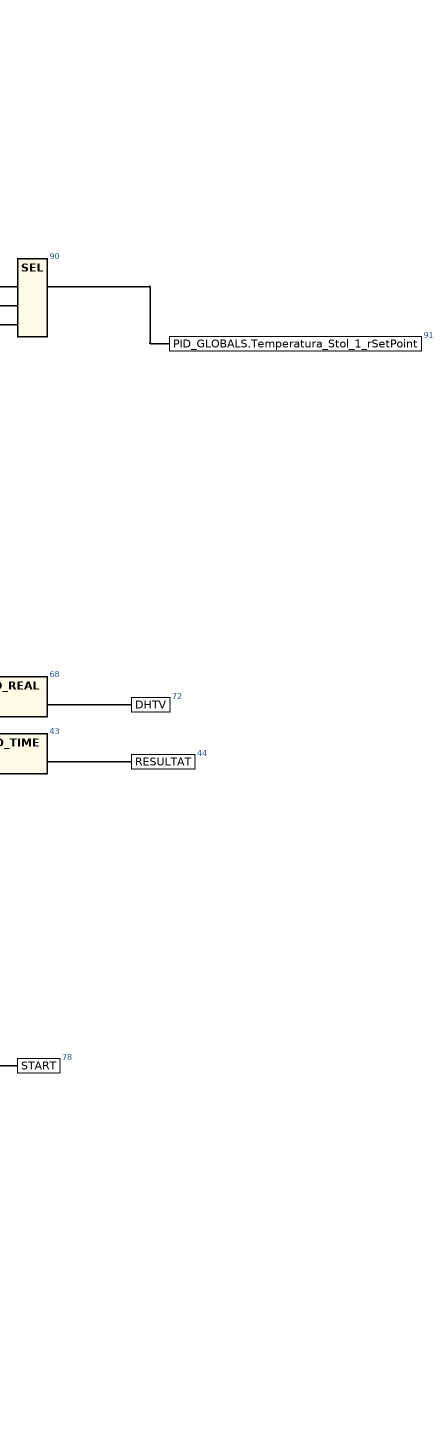
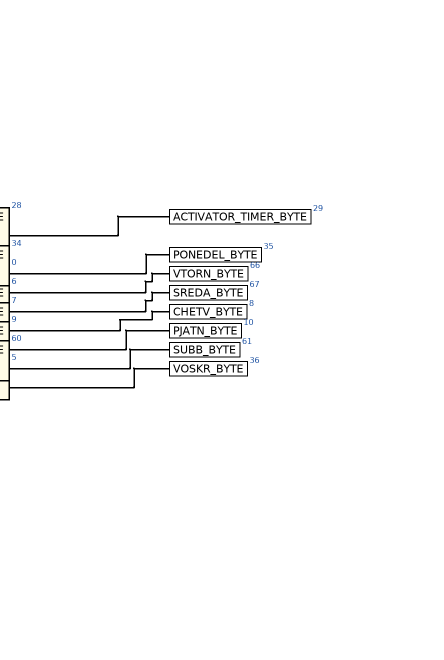
_w1 := BOOL_TO_BYTE(NVI_RETAIN.dateWeekStolOneTwo.2);
_w2 := HX3 * 60 + MX3;
Y4 := Y1;
X3 := _w2;
_w3 := BOOL_TO_BYTE(NVI_RETAIN.dateWeekStolOneTwo.3);
CHETV_BYTE := BOOL_TO_BYTE(NVI_RETAIN.dateWeekStolOneTwo.4);
PJATN_BYTE := BOOL_TO_BYTE(NVI_RETAIN.dateWeekStolOneTwo.5);
_w4 := GVL.hour = NVI_RETAIN.hourSundayStolOne;
_w5 := SEL(NVI_RETAIN.dateWeekStolOneTwo.4, 0, 4);
arrHist1[1] := Y2;
arrHist1[2] := Y3;
arrHist1[3] := Y4;
_w6 := GVL.hour = NVI_RETAIN.hourMondayStolOne;
_w7 := GVL.minute = NVI_RETAIN.minuteThursdayStolOne;
_w8 := GVL.minute = NVI_RETAIN.minuteFridayStolOne;
_w9 := GVL.minute = NVI_RETAIN.minuteSaturdayStolOne;
_w10 := GVL.minute = NVI_RETAIN.minuteTuesdayStolOne;
_w11 := GVL.day_of_week = SEL(NVI_RETAIN.dateWeekStolOneTwo.2, 0, 2);
_w12 := GVL.hour = NVI_RETAIN.hourThursdayStolOne;
ACTIVATOR_TIMER_BYTE := BOOL_TO_BYTE(NVI_RETAIN.dateWeekStolOneTwo.0);
_w13 := GVL.hour = NVI_RETAIN.hourFridayStolOne;
_w14 := GVL.hour = NVI_RETAIN.hourSaturdayStolOne;
_w15 := GVL.minute = NVI_RETAIN.minuteSundayStolOne;
_w16 := GVL.hour = NVI_RETAIN.hourWednesdayStolOne AND GVL.minute = NVI_RETAIN.minuteWednesdayStolOne AND GVL.day_of_week = SEL(NVI_RETAIN.dateWeekStolOneTwo.3, 0, 3);
PONEDEL_BYTE := BOOL_TO_BYTE(NVI_RETAIN.dateWeekStolOneTwo.1);
VOSKR_BYTE := BOOL_TO_BYTE(NVI_RETAIN.dateWeekStolOneTwo.7);
_w17 := HX2 * 60 + MX2;
RES := REAL_TO_TIME((_w17 + _w2) * 60000);
RESULTAT := REAL_TO_TIME(DHTV);
R_TRIG_02(CLK := STOP); // R_TRIG
_w18 := GVL.hour = NVI_RETAIN.hourTuesdayStolOne AND _w10 AND _w11;
arrHist1[0] := Y1;
R_TRIG_01(CLK := START); // R_TRIG
_w19 := X1 + X2;
_w20 := _w19 + X3;
_w21 := _w20 + X4;
SUBB_BYTE := BOOL_TO_BYTE(NVI_RETAIN.dateWeekStolOneTwo.6);
VTORN_BYTE := _w1;
SREDA_BYTE := _w3;
X2 := _w17;
DHTV := TIME_TO_REAL(T#1H25M);
R_TRIG_03(CLK := NVI_RETAIN.dateWeekStolOneTwo.0 AND (_w6 AND GVL.minute = NVI_RETAIN.minuteMondayStolOne AND GVL.day_of_week = SEL(NVI_RETAIN.dateWeekStolOneTwo.1, 0, 1) OR _w18 OR _w16 OR _w12 AND _w7 AND GVL.day_of_week = _w5 OR _w13 AND _w8 AND GVL.day_of_week = SEL(NVI_RETAIN.dateWeekStolOneTwo.5, 0, 5) OR _w14 AND _w9 AND GVL.day_of_week = SEL(NVI_RETAIN.dateWeekStolOneTwo.6, 0, 6) OR _w4 AND _w15 AND GVL.day_of_week = SEL(NVI_RETAIN.dateWeekStolOneTwo.7, 0, 7))); // R_TRIG
START := R_TRIG_03.Q;
RS_01(SET := R_TRIG_01.Q, RESET1 := _w22); // RS
_w23 := SEL(RS_01.Q1, 0, X);
INDIKATOR := RS_01.Q1;
TON1(IN := RS_01.Q1, PT := RES); // TON
_w22 := R_TRIG_02.Q OR TON1.Q;
ostanovka := _w22;
X := REAL_TO_INT(TIME_TO_REAL(TON1.ET) / 60000);
GR1(x := _w23, n := 4, x1 := X1, y1 := Y1, x2 := _w19, y2 := Y2, x3 := _w20, y3 := Y3, x4 := _w21, y4 := Y4); // GRAPH
PID_GLOBALS.Temperatura_Stol_1_rSetPoint := SEL(INDIKATOR, Y1, GR1.GRAPH1);

END_PROGRAM

// Device/Application/Parostol_Zadanie/GRAPH
(* @NESTEDCOMMENTS := 'Yes' *)
(* @PATH := '\/Доп. функции' *)
(* @OBJECTFLAGS := '0, 8' *)
(* @SYMFILEFLAGS := '2048' *)
FUNCTION_BLOCK GRAPH
VAR_INPUT
	x 	:REAL;
	n	:BYTE := 10;
	sort:BOOL;
	x1,y1,x2,y2,x3,y3,x4,y4(*,x5,y5,x6,y6,x7,y7,x8,y8,x9,y9,x10,y10*) :REAL;
	END_VAR
	VAR_OUTPUT
		GRAPH1:REAL;
	END_VAR

VAR
	i,j	:BYTE;
	swx,
	swy	:REAL;
	mini:BYTE;
	f	:BOOL;
	xy	:ARRAY[1..2,1..10] OF REAL;
	
END_VAR

(* @END_DECLARATION := '0' *)
xy[1,1]:=x1;
xy[1,2]:=x2;
xy[1,3]:=x3;
xy[1,4]:=x4;
//xy[1,5]:=x5;
//xy[1,6]:=x6;
//xy[1,7]:=x7;
//xy[1,8]:=x8;
//xy[1,9]:=x9;
//xy[1,10]:=x10;

xy[2,1]:=y1;
xy[2,2]:=y2;
xy[2,3]:=y3;
xy[2,4]:=y4;
//xy[2,5]:=y5;
//xy[2,6]:=y6;
//xy[2,7]:=y7;
//xy[2,8]:=y8;
//xy[2,9]:=y9;
//xy[2,10]:=y10;

IF sort THEN
	FOR j:=1 TO n DO
		f := FALSE; mini := j;
		FOR i:=j TO n-j DO
			IF xy[1,i] > xy[1,i+1] THEN
				swx:= xy[1,i]; swy:= xy[2,i];
				xy[1,i] := xy[1,i+1]; xy[2,i] := xy[2,i+1];
				xy[1,i+1] := swx; xy[2,i+1] := swy;
				f := TRUE;
			END_IF
			IF xy[1,i] < xy[1,mini] THEN mini := i; END_IF
		END_FOR
		IF NOT F THEN EXIT; END_IF
		IF mini <> j THEN
			swx:= xy[1,j]; swy:= xy[2,j];
			xy[1,j] := xy[1,mini]; xy[2,j] := xy[2,mini];
			xy[1,mini] := swx; xy[2,mini] := swy;
		END_IF
	END_FOR
END_IF

IF x < xy[1,1] THEN GRAPH1 := xy[2,1];
ELSIF x > xy[1,n] THEN GRAPH1 := xy[2,n];
ELSE
	FOR i:=1 TO n-1 DO
		IF x >= xy[1,i] AND x < xy[1,i+1] THEN
			GRAPH1 := (x-xy[1,i])*(xy[2,i+1]-xy[2,i])/(xy[1,i+1]-xy[1,i]) + xy[2,i];
		END_IF
	END_FOR
END_IF

END_FUNCTION_BLOCK

// Device/Application/Parostol_Zadanie/PLC_PRG_Stol_2
PROGRAM PLC_PRG_Stol_2
VAR
	
	TON1: TON;
	X: REAL;
	X1: BYTE:=1;

	X2: REAL;
	X3: REAL;
	X4: BYTE:=1;
	Y4: REAL;
	
	STOP: BOOL;			//
	
	GR1: GRAPH;
	
	arrHist1:ARRAY [0..3] OF REAL;
	
	DHTV: REAL;
	RESULTAT: TIME;
	RES: TIME;
	RS_01: RS;
	R_TRIG_01: R_TRIG;
	INDIKATOR: BOOL;
	R_TRIG_02: R_TRIG;
	R_TRIG_03: R_TRIG;
END_VAR

VAR RETAIN
	
	START: BOOL;
	
	Y1: REAL; 			//Начальная температу
	Y2: REAL;			//Температура подъёма
	Y3: REAL;			//Температура выдержки
	
	HX2: REAL;			//Время подъёма часы
	MX2: REAL;			//Время подъёма минуты
	HX3: REAL;			//Время выдержки часы
	MX3: REAL;			//Время выдержки минуты
	
	ACTIVATOR_TIMER: BOOL;//Активирование таймера
	//Понедельник
	PONEDEL:BOOL;
	HOUR_PONEDEL: BYTE;
	MINUTE_PONEDEL: BYTE;
	//Вторник
	VTORN:BOOL;	
	HOUR_VTORN: BYTE;
	MINUTE_VTORN: BYTE;
	//Среда
	SREDA: BOOL;
	HOUR_SREDA: BYTE;
	MINUTE_SREDA: BYTE;
	//Четверг
	CHETV: BOOL;
	HOUR_CHETV: BYTE;
	MINUTE_CHETV: BYTE;
	//Пятница
	PJATN: BOOL;
	HOUR_PJATN: BYTE;
	MINUTE_PJATN: BYTE;
	//Суббота
	SUBB: BOOL;
	HOUR_SUBB: BYTE;
	MINUTE_SUBB: BYTE;
	//Воскресенье
	VOSKR: BOOL;
	HOUR_VOSKR: BYTE;
	MINUTE_VOSKR: BYTE;
END_VAR
VAR // added by the converter: edge detectors and wires of the graphical bodies
    _w1, _w15, _w21 : REAL;
    _w2, _w4, _w5, _w6, _w7, _w8, _w9, _w10, _w11, _w12, _w13, _w14, _w16 : BOOL;
    _w3, _w20 : ANY;
    _w17, _w18, _w19 : BYTE;
END_VAR

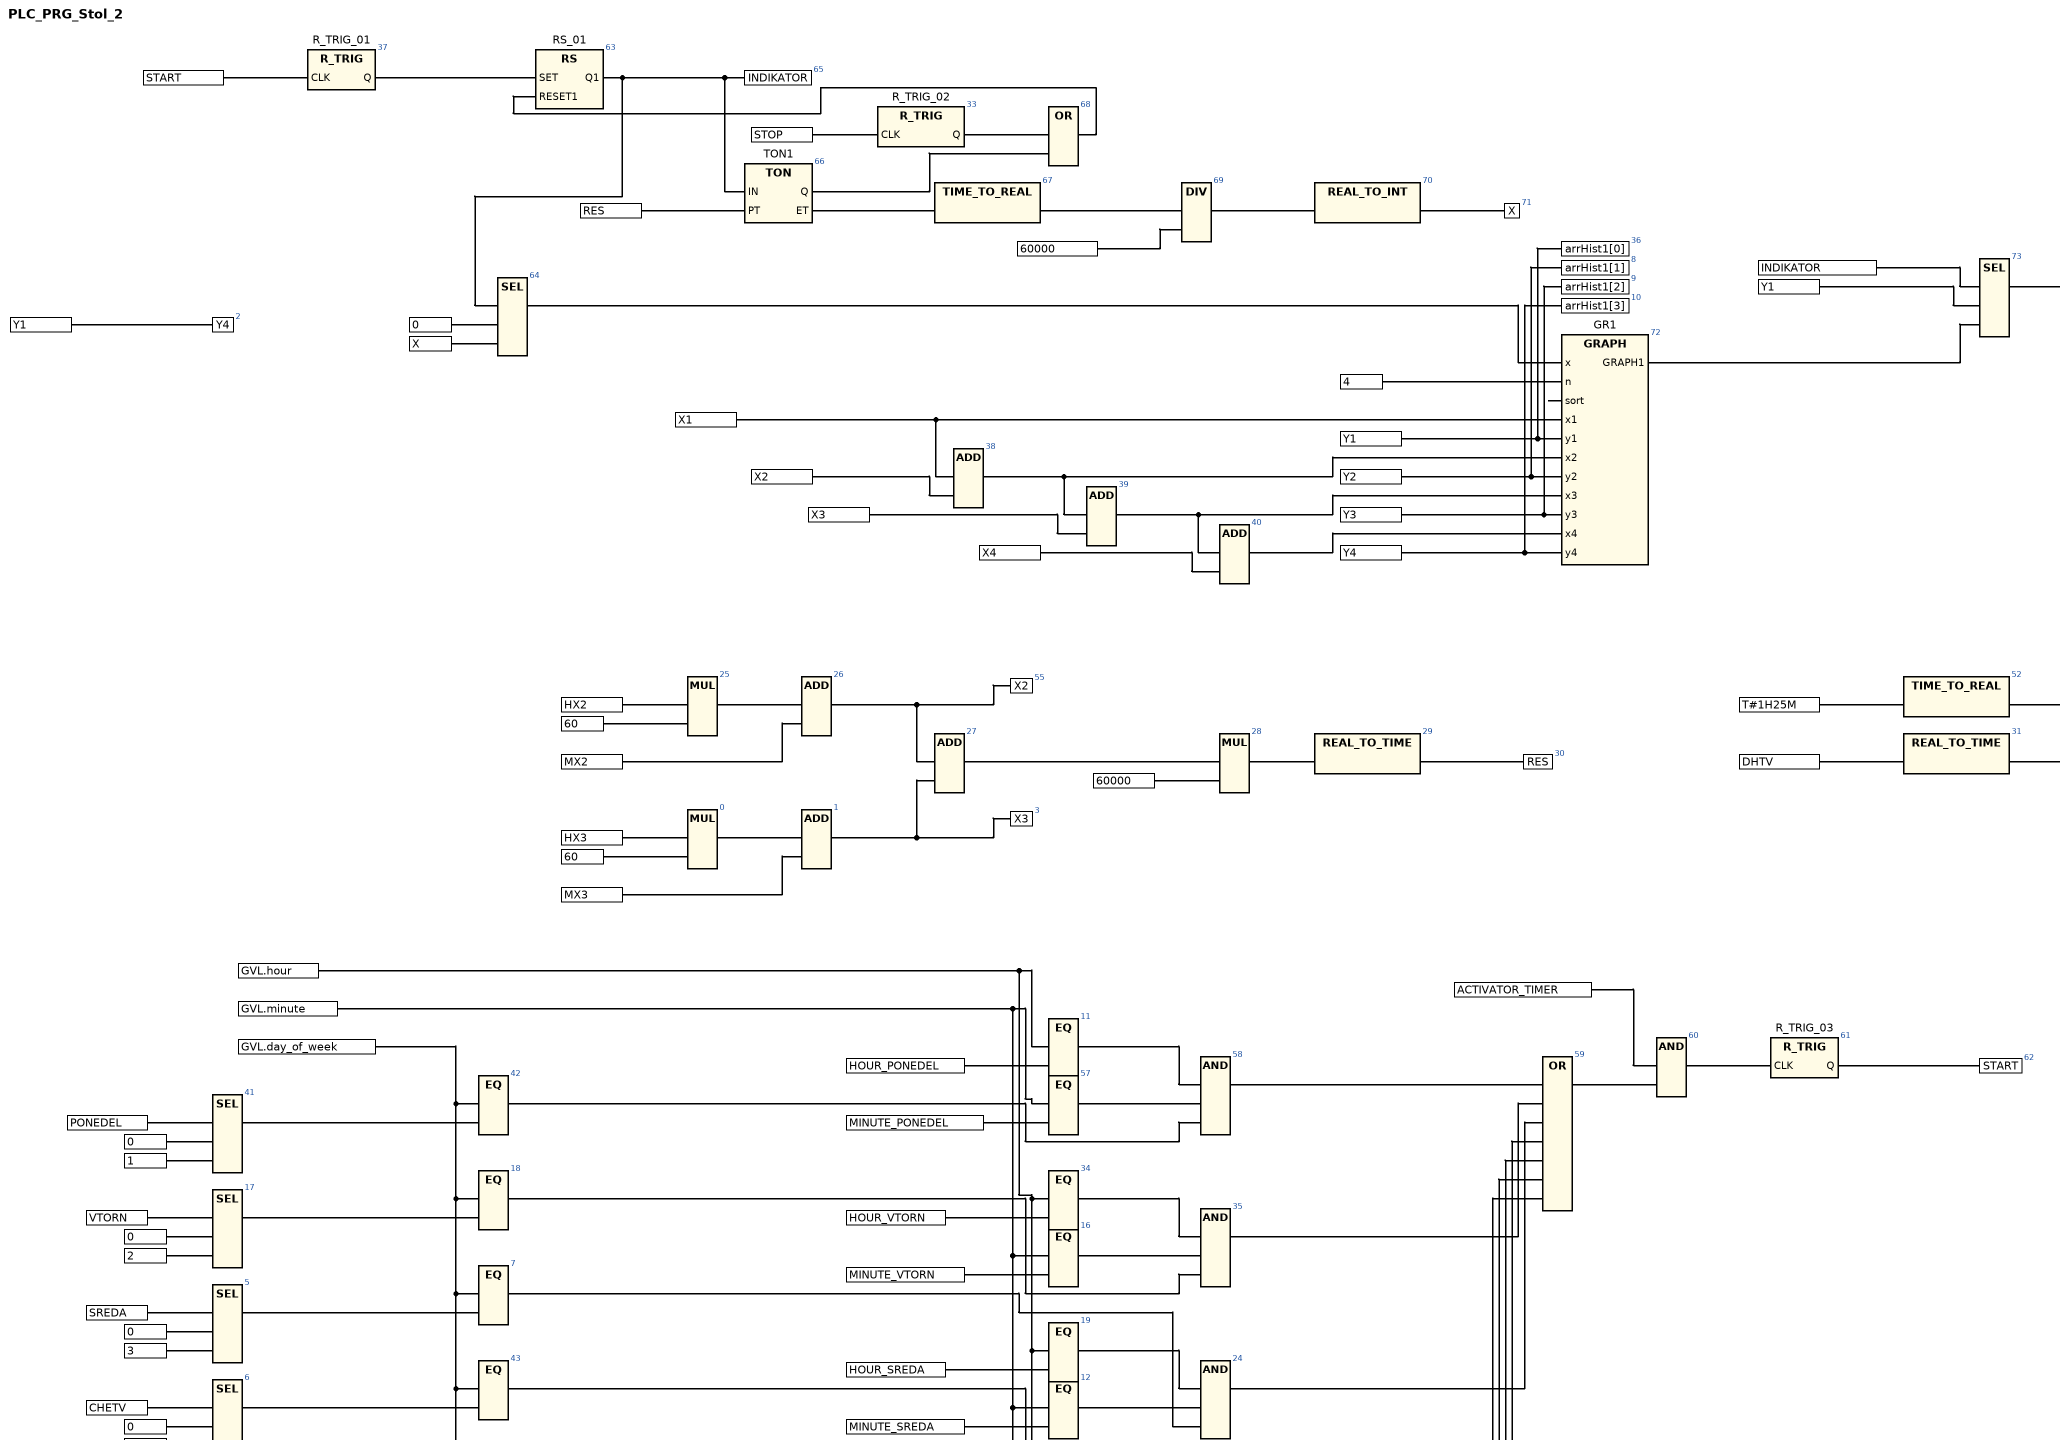
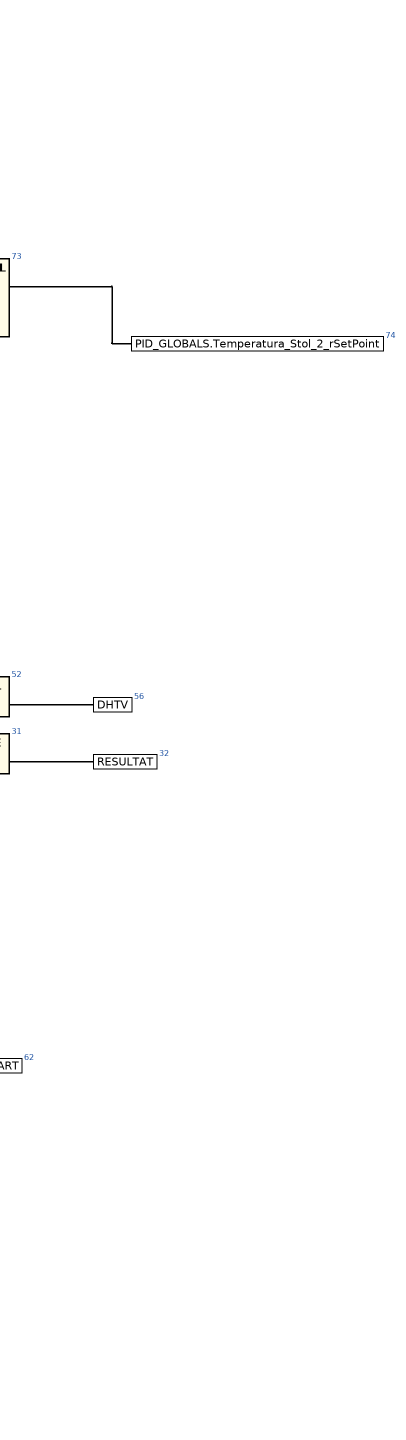
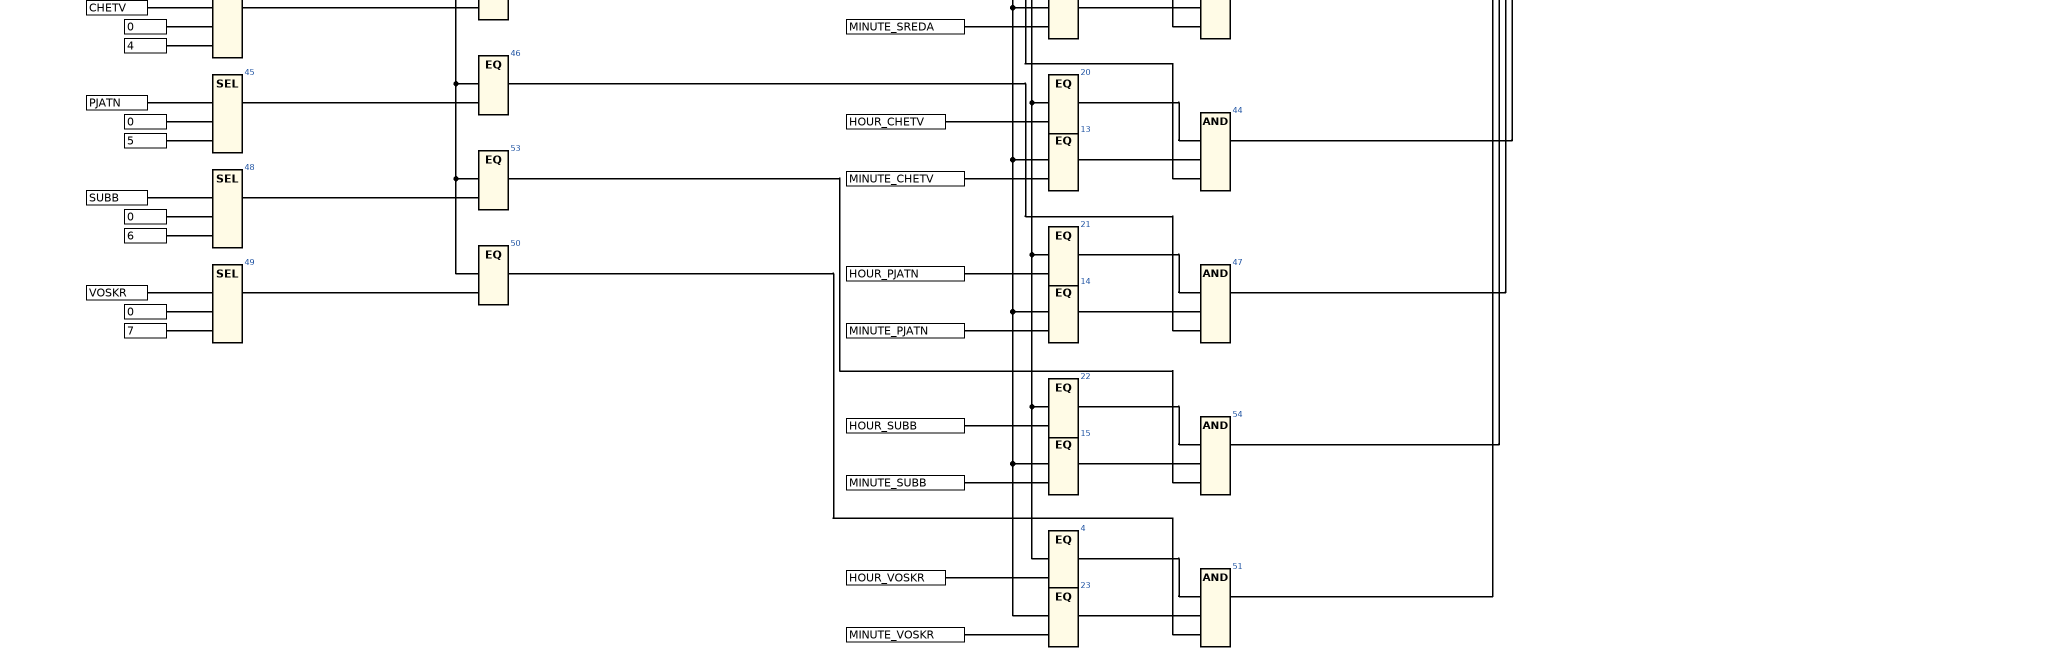
_w1 := HX3 * 60 + MX3;
Y4 := Y1;
X3 := _w1;
_w2 := GVL.hour = HOUR_VOSKR;
_w3 := SEL(CHETV, 0, 4);
arrHist1[1] := Y2;
arrHist1[2] := Y3;
arrHist1[3] := Y4;
_w4 := GVL.hour = HOUR_PONEDEL;
_w5 := GVL.minute = MINUTE_CHETV;
_w6 := GVL.minute = MINUTE_PJATN;
_w7 := GVL.minute = MINUTE_SUBB;
_w8 := GVL.minute = MINUTE_VTORN;
_w9 := GVL.day_of_week = SEL(VTORN, 0, 2);
_w10 := GVL.hour = HOUR_CHETV;
_w11 := GVL.hour = HOUR_PJATN;
_w12 := GVL.hour = HOUR_SUBB;
_w13 := GVL.minute = MINUTE_VOSKR;
_w14 := GVL.hour = HOUR_SREDA AND GVL.minute = MINUTE_SREDA AND GVL.day_of_week = SEL(SREDA, 0, 3);
_w15 := HX2 * 60 + MX2;
RES := REAL_TO_TIME((_w15 + _w1) * 60000);
RESULTAT := REAL_TO_TIME(DHTV);
R_TRIG_02(CLK := STOP); // R_TRIG
_w16 := GVL.hour = HOUR_VTORN AND _w8 AND _w9;
arrHist1[0] := Y1;
R_TRIG_01(CLK := START); // R_TRIG
_w17 := X1 + X2;
_w18 := _w17 + X3;
_w19 := _w18 + X4;
X2 := _w15;
DHTV := TIME_TO_REAL(T#1H25M);
R_TRIG_03(CLK := ACTIVATOR_TIMER AND (_w4 AND GVL.minute = MINUTE_PONEDEL AND GVL.day_of_week = SEL(PONEDEL, 0, 1) OR _w16 OR _w14 OR _w10 AND _w5 AND GVL.day_of_week = _w3 OR _w11 AND _w6 AND GVL.day_of_week = SEL(PJATN, 0, 5) OR _w12 AND _w7 AND GVL.day_of_week = SEL(SUBB, 0, 6) OR _w2 AND _w13 AND GVL.day_of_week = SEL(VOSKR, 0, 7))); // R_TRIG
START := R_TRIG_03.Q;
RS_01(SET := R_TRIG_01.Q, RESET1 := _w20); // RS
_w21 := SEL(RS_01.Q1, 0, X);
INDIKATOR := RS_01.Q1;
TON1(IN := RS_01.Q1, PT := RES); // TON
_w20 := R_TRIG_02.Q OR TON1.Q;
X := REAL_TO_INT(TIME_TO_REAL(TON1.ET) / 60000);
GR1(x := _w21, n := 4, x1 := X1, y1 := Y1, x2 := _w17, y2 := Y2, x3 := _w18, y3 := Y3, x4 := _w19, y4 := Y4); // GRAPH
PID_GLOBALS.Temperatura_Stol_2_rSetPoint := SEL(INDIKATOR, Y1, GR1.GRAPH1);

END_PROGRAM

// Device/Application/Parostol_Zadanie/PLC_PRG_Stol_3
PROGRAM PLC_PRG_Stol_3
VAR
	
	TON1: 							TON;
	X: 								REAL;
	X1: 							BYTE:=1;

	X2: 							REAL;
	X3: 							REAL;
	X4: 							BYTE:=1;
	Y4: 							REAL;
	GR1: 							GRAPH;
	
	arrHist1:						ARRAY [0..3] OF REAL;
	
	DHTV: 							REAL;
	RESULTAT: 						TIME;
	RES: 							TIME;
	RS_01: 							RS;
	R_TRIG_01: 						R_TRIG;
	INDIKATOR: 						BOOL;
	R_TRIG_02: 						R_TRIG;
	STOP: 							BOOL;
	R_TRIG_03: 						R_TRIG;
	
	// Конвертация для архивации
	ACTIVATOR_TIMER_BYTE:		BYTE;
	PONEDEL_BYTE:				BYTE;					
	VTORN_BYTE:					BYTE;		
	SREDA_BYTE:					BYTE;
	CHETV_BYTE:					BYTE;
	PJATN_BYTE:					BYTE;
	SUBB_BYTE:					BYTE;
	VOSKR_BYTE:					BYTE;
	
	ostanovka: 					BOOL;						// Переменная для команды запуска закрытия 3-х ходового
END_VAR

VAR RETAIN
	
	START: 							BOOL;
	
	Y1: 							REAL; 					// Начальная температу
	Y2: 							REAL;					// Температура подъёма
	Y3: 							REAL;					// Температура выдержки
	
	HX2: 							REAL;					// Время подъёма минуты
	MX2: 							REAL;					// Время подъёма минуты
	HX3: 							REAL;					// Время выдержки часы
	MX3: 							REAL;					// Время выдержки минуты
END_VAR
VAR // added by the converter: edge detectors and wires of the graphical bodies
    _w1, _w18, _w19, _w20 : BYTE;
    _w2, _w16, _w22 : REAL;
    _w3, _w5, _w6, _w7, _w8, _w9, _w10, _w11, _w12, _w13, _w14, _w15, _w17 : BOOL;
    _w4, _w21 : ANY;
END_VAR

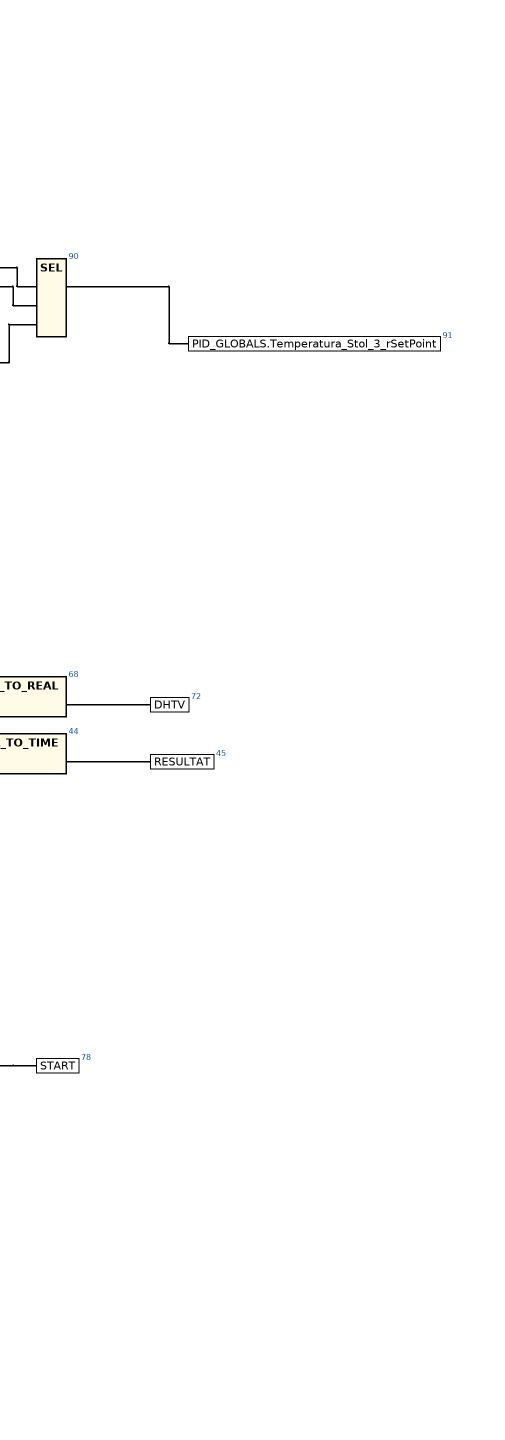
_w1 := BOOL_TO_BYTE(NVI_RETAIN.dateWeekStolThreeFour.6);
PONEDEL_BYTE := BOOL_TO_BYTE(NVI_RETAIN.dateWeekStolThreeFour.1);
_w2 := HX3 * 60 + MX3;
Y4 := Y1;
X3 := _w2;
_w3 := GVL.hour = NVI_RETAIN.hourSundayStolThree;
_w4 := SEL(NVI_RETAIN.dateWeekStolThreeFour.4, 0, 4);
ACTIVATOR_TIMER_BYTE := BOOL_TO_BYTE(NVI_RETAIN.dateWeekStolThreeFour.0);
arrHist1[1] := Y2;
arrHist1[2] := Y3;
arrHist1[3] := Y4;
// Для запуска работы по времени
_w5 := GVL.hour = NVI_RETAIN.hourMondayStolThree;
_w6 := GVL.minute = NVI_RETAIN.minuteThursdayStolThree;
SREDA_BYTE := BOOL_TO_BYTE(NVI_RETAIN.dateWeekStolThreeFour.3);
PJATN_BYTE := BOOL_TO_BYTE(NVI_RETAIN.dateWeekStolThreeFour.5);
CHETV_BYTE := BOOL_TO_BYTE(NVI_RETAIN.dateWeekStolThreeFour.4);
_w7 := GVL.minute = NVI_RETAIN.minuteFridayStolThree;
_w8 := GVL.minute = NVI_RETAIN.minuteSaturdayStolThree;
_w9 := GVL.minute = NVI_RETAIN.minuteTuesdayStolThree;
_w10 := GVL.day_of_week = SEL(NVI_RETAIN.dateWeekStolThreeFour.2, 0, 2);
_w11 := GVL.hour = NVI_RETAIN.hourThursdayStolThree;
VTORN_BYTE := BOOL_TO_BYTE(NVI_RETAIN.dateWeekStolThreeFour.2);
_w12 := GVL.hour = NVI_RETAIN.hourFridayStolThree;
_w13 := GVL.hour = NVI_RETAIN.hourSaturdayStolThree;
_w14 := GVL.minute = NVI_RETAIN.minuteSundayStolThree;
_w15 := GVL.hour = NVI_RETAIN.hourWednesdayStolThree AND GVL.minute = NVI_RETAIN.minuteWednesdayStolThree AND GVL.day_of_week = SEL(NVI_RETAIN.dateWeekStolThreeFour.3, 0, 3);
_w16 := HX2 * 60 + MX2;
RES := REAL_TO_TIME((_w16 + _w2) * 60000);
RESULTAT := REAL_TO_TIME(DHTV);
R_TRIG_02(CLK := STOP); // R_TRIG
_w17 := GVL.hour = NVI_RETAIN.hourTuesdayStolThree AND _w9 AND _w10;
arrHist1[0] := Y1;
R_TRIG_01(CLK := START); // R_TRIG
_w18 := X1 + X2;
_w19 := _w18 + X3;
_w20 := _w19 + X4;
VOSKR_BYTE := BOOL_TO_BYTE(NVI_RETAIN.dateWeekStolThreeFour.7);
SUBB_BYTE := _w1;
X2 := _w16;
DHTV := TIME_TO_REAL(T#1H25M);
R_TRIG_03(CLK := NVI_RETAIN.dateWeekStolThreeFour.0 AND (_w5 AND GVL.minute = NVI_RETAIN.minuteMondayStolThree AND GVL.day_of_week = SEL(NVI_RETAIN.dateWeekStolThreeFour.1, 0, 1) OR _w17 OR _w15 OR _w11 AND _w6 AND GVL.day_of_week = _w4 OR _w12 AND _w7 AND GVL.day_of_week = SEL(NVI_RETAIN.dateWeekStolThreeFour.5, 0, 5) OR _w13 AND _w8 AND GVL.day_of_week = SEL(NVI_RETAIN.dateWeekStolThreeFour.6, 0, 6) OR _w3 AND _w14 AND GVL.day_of_week = SEL(NVI_RETAIN.dateWeekStolThreeFour.7, 0, 7))); // R_TRIG
START := R_TRIG_03.Q;
RS_01(SET := R_TRIG_01.Q, RESET1 := _w21); // RS
_w22 := SEL(RS_01.Q1, 0, X);
INDIKATOR := RS_01.Q1;
TON1(IN := RS_01.Q1, PT := RES); // TON
_w21 := R_TRIG_02.Q OR TON1.Q;
ostanovka := _w21;
X := REAL_TO_INT(TIME_TO_REAL(TON1.ET) / 60000);
GR1(x := _w22, n := 4, x1 := X1, y1 := Y1, x2 := _w18, y2 := Y2, x3 := _w19, y3 := Y3, x4 := _w20, y4 := Y4); // GRAPH
PID_GLOBALS.Temperatura_Stol_3_rSetPoint := SEL(INDIKATOR, Y1, GR1.GRAPH1);

END_PROGRAM

// Device/Application/Parostol_Zadanie/PLC_PRG_Stol_4
PROGRAM PLC_PRG_Stol_4
VAR
	
	TON1: 						TON;
	X: 							REAL;
	X1: 						BYTE:=1;

	X2: 						REAL;
	X3: 						REAL;
	X4: 						BYTE:=1;
	Y4: 						REAL;
	GR1: 						GRAPH;
	
	arrHist1:					ARRAY [0..3] OF REAL;
	
	DHTV: 						REAL;
	RESULTAT:					TIME;
	RES: 						TIME;
	RS_01: 						RS;
	R_TRIG_01: 					R_TRIG;
	INDIKATOR: 					BOOL;
	R_TRIG_02: 					R_TRIG;
	STOP: 						BOOL;
	R_TRIG_03: 					R_TRIG;
	
	// Конвертация для архивации
	ACTIVATOR_TIMER_BYTE:		BYTE;
	PONEDEL_BYTE:				BYTE;					
	VTORN_BYTE:					BYTE;		
	SREDA_BYTE:					BYTE;
	CHETV_BYTE:					BYTE;
	PJATN_BYTE:					BYTE;
	SUBB_BYTE:					BYTE;
	VOSKR_BYTE:					BYTE;
	ostanovka: 					BOOL;						// Переменная для команды запуска закрытия 3-х ходового
END_VAR

VAR RETAIN
	
	START: 						BOOL;
	
	Y1: 						REAL; 					// Начальная температу
	Y2: 						REAL;					// Температура подъёма
	Y3: 						REAL;					// Температура выдержки
	
	HX2: 						REAL;					// Время подъёма часы
	MX2: 						REAL;					// Время подъёма минуты
	HX3: 						REAL;					// Время выдержки часы
	MX3: 						REAL;					// Время выдержки минуты
END_VAR
VAR // added by the converter: edge detectors and wires of the graphical bodies
    _w1, _w16, _w22 : REAL;
    _w2, _w4, _w6, _w7, _w8, _w9, _w10, _w11, _w12, _w13, _w14, _w15, _w17 : BOOL;
    _w3, _w21 : ANY;
    _w5, _w18, _w19, _w20 : BYTE;
END_VAR

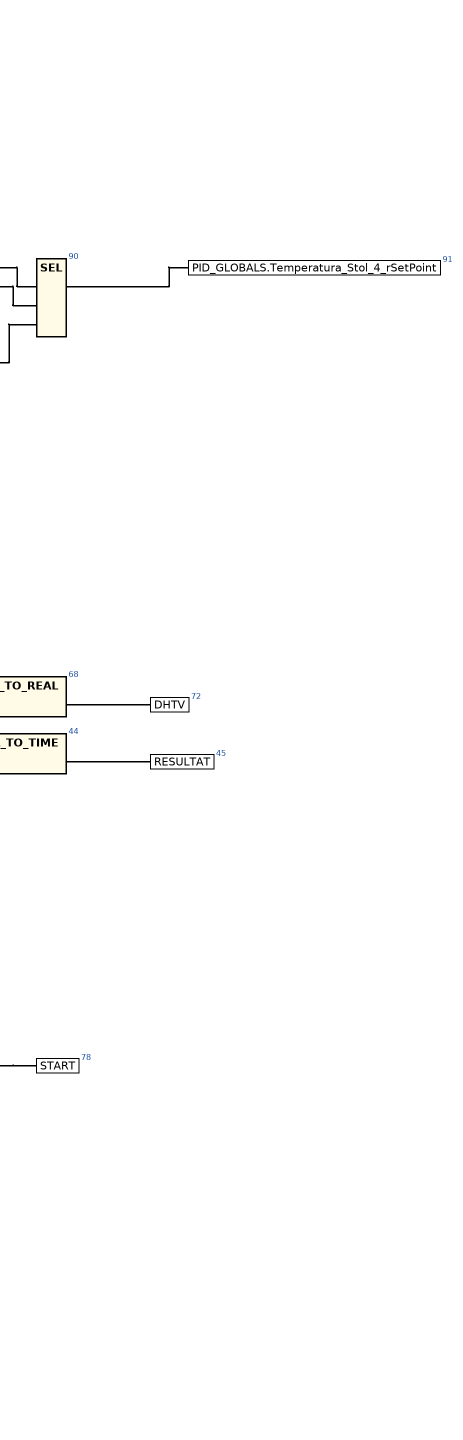
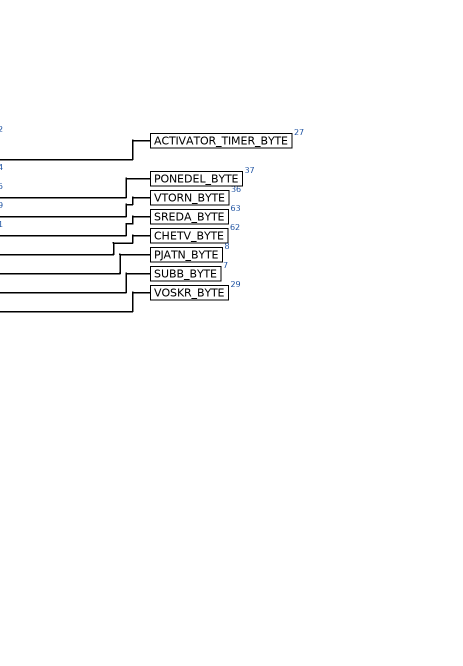
_w1 := HX3 * 60 + MX3;
Y4 := Y1;
X3 := _w1;
SUBB_BYTE := BOOL_TO_BYTE(NVI_RETAIN.dateWeekStolThreeFour.14);
PJATN_BYTE := BOOL_TO_BYTE(NVI_RETAIN.dateWeekStolThreeFour.13);
_w2 := GVL.hour = NVI_RETAIN.hourSundayStolFour;
_w3 := SEL(NVI_RETAIN.dateWeekStolThreeFour.12, 0, 4);
arrHist1[1] := Y2;
arrHist1[2] := Y3;
arrHist1[3] := Y4;
_w4 := GVL.hour = NVI_RETAIN.hourMondayStolFour;
_w5 := BOOL_TO_BYTE(NVI_RETAIN.dateWeekStolThreeFour.11);
_w6 := GVL.minute = NVI_RETAIN.minuteThursdayStolFour;
_w7 := GVL.minute = NVI_RETAIN.minuteFridayStolFour;
_w8 := GVL.minute = NVI_RETAIN.minuteSaturdayStolFour;
_w9 := GVL.minute = NVI_RETAIN.minuteTuesdayStolFour;
_w10 := GVL.day_of_week = SEL(NVI_RETAIN.dateWeekStolThreeFour.10, 0, 2);
ACTIVATOR_TIMER_BYTE := BOOL_TO_BYTE(NVI_RETAIN.dateWeekStolThreeFour.8);
_w11 := GVL.hour = NVI_RETAIN.hourThursdayStolFour;
VOSKR_BYTE := BOOL_TO_BYTE(NVI_RETAIN.dateWeekStolThreeFour.15);
_w12 := GVL.hour = NVI_RETAIN.hourFridayStolFour;
_w13 := GVL.hour = NVI_RETAIN.hourSaturdayStolFour;
_w14 := GVL.minute = NVI_RETAIN.minuteSundayStolFour;
_w15 := GVL.hour = NVI_RETAIN.hourWednesdayStolFour AND GVL.minute = NVI_RETAIN.minuteWednesdayStolFour AND GVL.day_of_week = SEL(NVI_RETAIN.dateWeekStolThreeFour.11, 0, 3);
VTORN_BYTE := BOOL_TO_BYTE(NVI_RETAIN.dateWeekStolThreeFour.10);
PONEDEL_BYTE := BOOL_TO_BYTE(NVI_RETAIN.dateWeekStolThreeFour.9);
_w16 := HX2 * 60 + MX2;
RES := REAL_TO_TIME((_w16 + _w1) * 60000);
RESULTAT := REAL_TO_TIME(DHTV);
R_TRIG_02(CLK := STOP); // R_TRIG
_w17 := GVL.hour = NVI_RETAIN.hourTuesdayStolFour AND _w9 AND _w10;
arrHist1[0] := Y1;
R_TRIG_01(CLK := START); // R_TRIG
_w18 := X1 + X2;
_w19 := _w18 + X3;
_w20 := _w19 + X4;
CHETV_BYTE := BOOL_TO_BYTE(NVI_RETAIN.dateWeekStolThreeFour.12);
SREDA_BYTE := _w5;
X2 := _w16;
DHTV := TIME_TO_REAL(T#1H25M);
R_TRIG_03(CLK := NVI_RETAIN.dateWeekStolThreeFour.8 AND (_w4 AND GVL.minute = NVI_RETAIN.minuteMondayStolFour AND GVL.day_of_week = SEL(NVI_RETAIN.dateWeekStolThreeFour.9, 0, 1) OR _w17 OR _w15 OR _w11 AND _w6 AND GVL.day_of_week = _w3 OR _w12 AND _w7 AND GVL.day_of_week = SEL(NVI_RETAIN.dateWeekStolThreeFour.13, 0, 5) OR _w13 AND _w8 AND GVL.day_of_week = SEL(NVI_RETAIN.dateWeekStolThreeFour.14, 0, 6) OR _w2 AND _w14 AND GVL.day_of_week = SEL(NVI_RETAIN.dateWeekStolThreeFour.15, 0, 7))); // R_TRIG
START := R_TRIG_03.Q;
RS_01(SET := R_TRIG_01.Q, RESET1 := _w21); // RS
_w22 := SEL(RS_01.Q1, 0, X);
INDIKATOR := RS_01.Q1;
TON1(IN := RS_01.Q1, PT := RES); // TON
_w21 := R_TRIG_02.Q OR TON1.Q;
ostanovka := _w21;
X := REAL_TO_INT(TIME_TO_REAL(TON1.ET) / 60000);
GR1(x := _w22, n := 4, x1 := X1, y1 := Y1, x2 := _w18, y2 := Y2, x3 := _w19, y3 := Y3, x4 := _w20, y4 := Y4); // GRAPH
PID_GLOBALS.Temperatura_Stol_4_rSetPoint := SEL(INDIKATOR, Y1, GR1.GRAPH1);

END_PROGRAM

// Device/Application/CFC_Davlenie_PID/PLC_PRG_CFC_Davlenie_Stol_1_2
PROGRAM PLC_PRG_CFC_Davlenie_Stol_1_2
VAR
	(* входы регулятора *)
	//
	fbApidPosValv: 							OPR.APID_POS_VALV;		// ФБ ПИД регулятора с АНР
	fbDy_manualTrig_r:						R_TRIG;					// Детектор нажатия кнопки записи мощности в ручном режиме на вход DY_MANUAL
	fbDy_manualTrig_f:						F_TRIG;					// Детектор отпускания кнопки для сброса входа DY_MANUAL в 0
	rCurrentValue: 							REAL;					// Измеренное значение регулируемой величины
	rDY_MANUAL: 							REAL;					// Мощность, передаваемая на вход DY_MANUAL
	wSampleTime_0:							WORD;					// Значение PV_TIME в предыдущем цикле ПЛК
	fbCountChangePV_TIME: 					CTU;					// Счетчик циклов ПЛК, в которых происходило изменение PV_TIME
	xSetSP: 								BOOL;					// Команда на запись SP
	xSetSPFirst: 							BOOL;					// Команда на запись SP при запуске контроллера
	xSetSPFirstFlag: 						BOOL	:=	TRUE;		// Флаг записи SP при запуске контроллера
	fbEnabledPidTrig_f: 					F_TRIG;					// Детектор импульса на запись уставки в первом цикле ПЛК
	(* выходы регулятора *)
	//
	ePidState: 								OPR.STATE_PID;			// Состояние регулятора
	ePidError: 								OPR.ERROR_PID;			// Код ошибки регулятора
	xLess: 									BOOL;					// Сигнал на закрытие ИМ
	xMore:									BOOL;					// Сигнал на открытие ИМ
	rYsm: 									REAL;					// Расчетное положение выхода задвижки (для аналогового управления)
	rYsm_scale: 							REAL;					// Расчетное положение выхода задвижки, отображаемое на тренде
	xDendh:									BOOL;					// Признак достижения задвижкой 100%
	xDendl:									BOOL;					// Признак достижения задвижкой 0%
	(* параметры АНР *)
	//
	eAutotuneMode: 							OPR.TYPE_ANR;			// Тип автонастройки  (DYNAMIC - быстрый переход на новую уставку, но возможно перерегулирование; STABILITY - медленный переход на новую уставку, но с меньшим перерегулирование)
	xStartAutotune:							BOOL;					// Команда запуска АНР
	xStartFirstAutotune:					BOOL;					// Команда автоматического запуска АНР при включении контроллера (при нулевых параметрах ПИД)
	fbAutotuneCompletedTrig:				R_TRIG;					// Детектор импульса завершения АНР
	fbSetSPAnr: 							R_TRIG;					// Детектор импульса на запись SP при запуске АНР
	(* параметры ручного управления *)
	//
	fbManualModeExited: 					F_TRIG;					// Детектор импульса выхода из режима ручного управления
	xManual_set:							BOOL;					// Команда записи мощности в ручном режиме
	rManual_mean: 							REAL;					// Значение передаваемой мощности в ручном режиме
	xSetManualOK:							BOOL;					// Сигнал, указывающий на возможность безударного включения ручного режима (сигнал отсутствия регулирования)
	fbDy_manualTrig_r_anr: 					R_TRIG;					// Детектор импульса включения ручного режима при активной АНР
	fbDy_manualTrig_f_anr: 					F_TRIG;					// Задержка на цикл ПЛК на передачу параметра на вход rDy_anr
	fbDy_manualTrig_f_anr_0: 				F_TRIG;					// Сброс входа rDy_anr
	(* запись параметров регулятора *)
	//	
	xWritePidSettingsAfterReboot: 			BOOL	:=	TRUE;		// Команда восстановления параметров ПИД после перезагрузки контроллера
	xWritePidSettings:						BOOL	:=	TRUE;		// Команда записи параметров ПИД, введенных пользователем
	fbWritePidSettingsTrig: 				R_TRIG;					// Детектор импульса записи параметров ПИД пользователем
	(* ФБ записи параметров *)
	//
	fbWritePidSettings: 					OPR.SET_APID_POS_VALV;	// ФБ записи параметров ПИД
	fbWritePidSettingsAfterRebootTrig:		R_TRIG;					// Детектор импульса записи параметров ПИД после перезагрузки контроллера
	(* ФБ чтения параметров *)
	//	
	fbReadPidSettings: 						OPR.GET_APID_POS_VALV;	// ФБ чтения параметров ПИД
	fbReadPidSettingsTrig: 					F_TRIG;					// Детектор импульса чтения параметров ПИД
	(* Параметры выходов ПЛК *)
	//
	(*Параметры сброса ФБ ПИД*)
	fbApidPosValvReset: 					OPR.APID_POS_VALV;		// ФБ ПИД регулятора, используемый для сброса параметров основного ФБ ПИД перед запуском АНР
	xReset: 								BOOL;					// Команда на сброс ФБ ПИД
	fbReset: 								R_TRIG;					// Детектор импульса от переменной xReset
	xFirstCycle:						 	BOOL	:=	TRUE;		// Команда на сброс ФБ ПИД после перезагрузки ПЛК, в случае ранее активной АНР или ручного режима
	fbOffReset: 							R_TRIG;					// Детектор импульса от переменной xFirstCucle

END_VAR
VAR RETAIN
	Davlenie_Stol_1_2_rSetPoint: 			REAL;					// Дельта давления
	xIsEnabledPid:							BOOL 	:= 	TRUE;		// Состояние регулятора (TRUE - включен)
	rTval: 									REAL	:=	120;		// Время полного хода ИМ, сек
	rTluft:									REAL	:=	0.0;		// Время выборки люфта ИМ, сек
	rTimp:									REAL	:=	5;		// Минимальная длительность импульса, сек
	rDy_anr: 								REAL	:=	50.0;		// Размах мощности,%
	rSetPoint: 								REAL	:=	0.35;		// Уставка регулятора
	rSteadyValue: 							REAL	:=	0.3;		// Значение регулируемого параметра при нулевой мощности управляющего сигнала 
	rDeadBand: 								REAL 	:=	0.03;		// Зона нечувствительности ПИД
	rZeroBandForPidParams:					REAL	:=	0.001;		// Зона нулевых коэффициентов ПИД
	//
	rXp: 									REAL:=2.85;					// Полоса пропускания (100/Кр)
	rTi: 									REAL:=7.56;					// Постоянная времени интегрирования
	rTd: 									REAL:=1.64;					// Постоянная времени дифференцирования
	rSpeedOutLimit: 						REAL;					// Допустимая скорость изменения внутренней уставки ПИД
	rFilterTime: 							REAL;					// Постоянная времени входного фильтра ПИД
	//										
	xAutotuneCompleted:						BOOL;					// Импульс завершения АНР
	xIsPidValidSettings: 					BOOL;					// Сигнал настройки ПИД
	xManualMode: 							BOOL;					// Сигнал перевода ПИД в режим ручного управления
	xAutotuneInProgress:					BOOL;					// Флаг "Выполняется АНР"
END_VAR
VAR // added by the converter: edge detectors and wires of the graphical bodies
    _w1, _w8, _w11, _w13, _w14, _w15, _w25, _w27 : ANY;
    _w2, _w3, _w5, _w9, _w10, _w12, _w16, _w18, _w19, _w20, _w21, _w22, _w23, _w24, _w26, _w28, _w29, _w30 : BOOL;
    _w4, _w6, _w17 : REAL;
    _w7 : OPR.APID_POS_VALV;
END_VAR

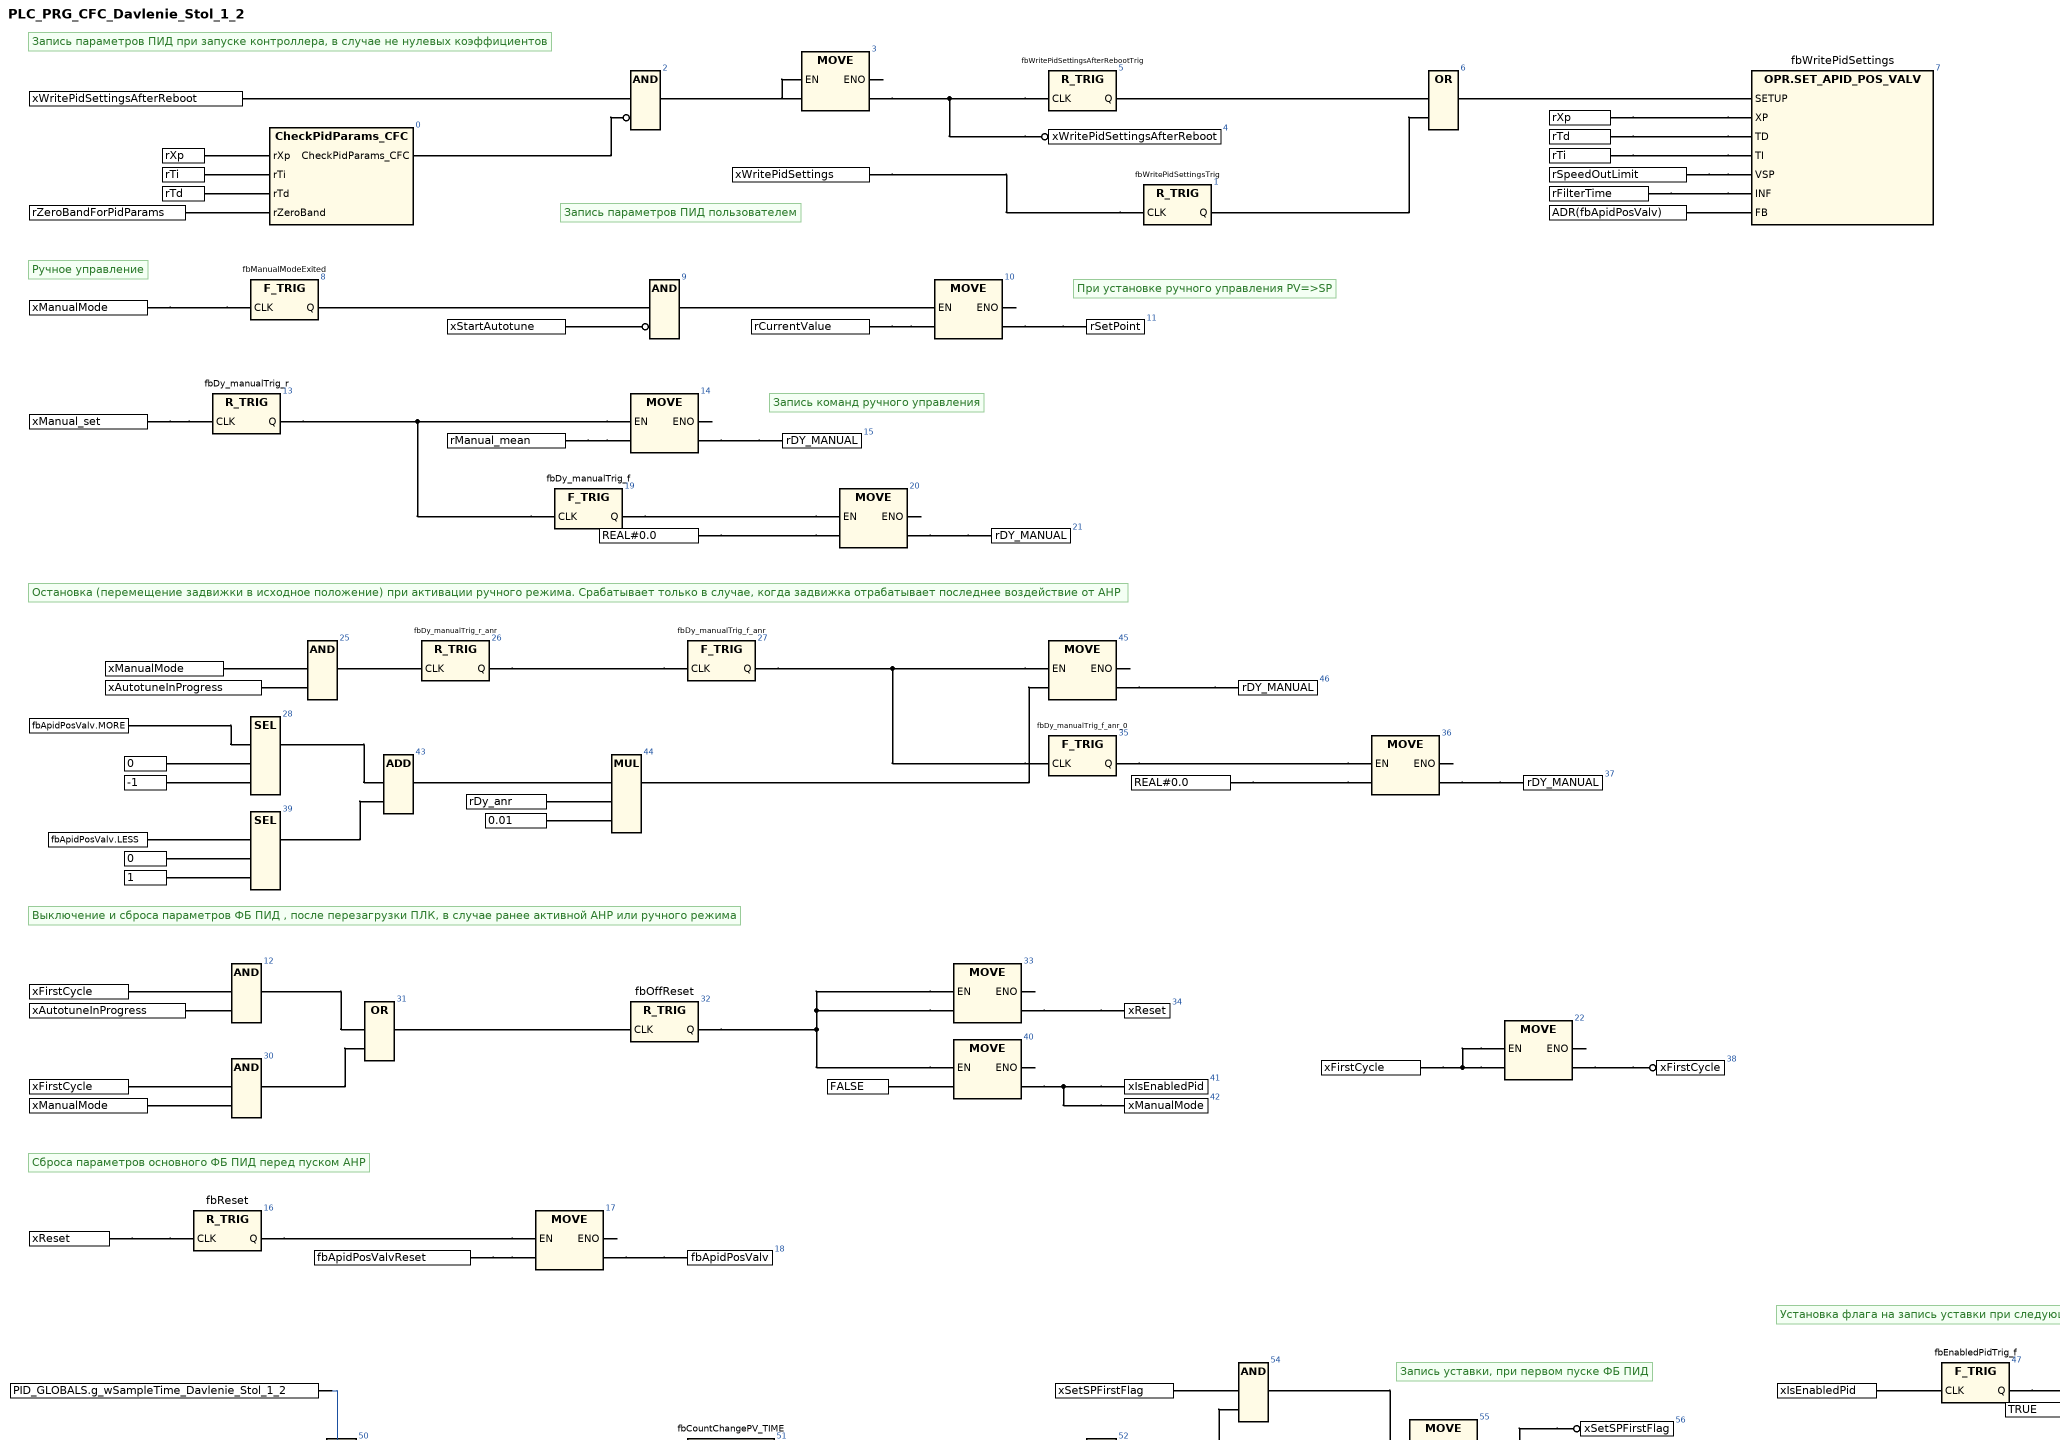
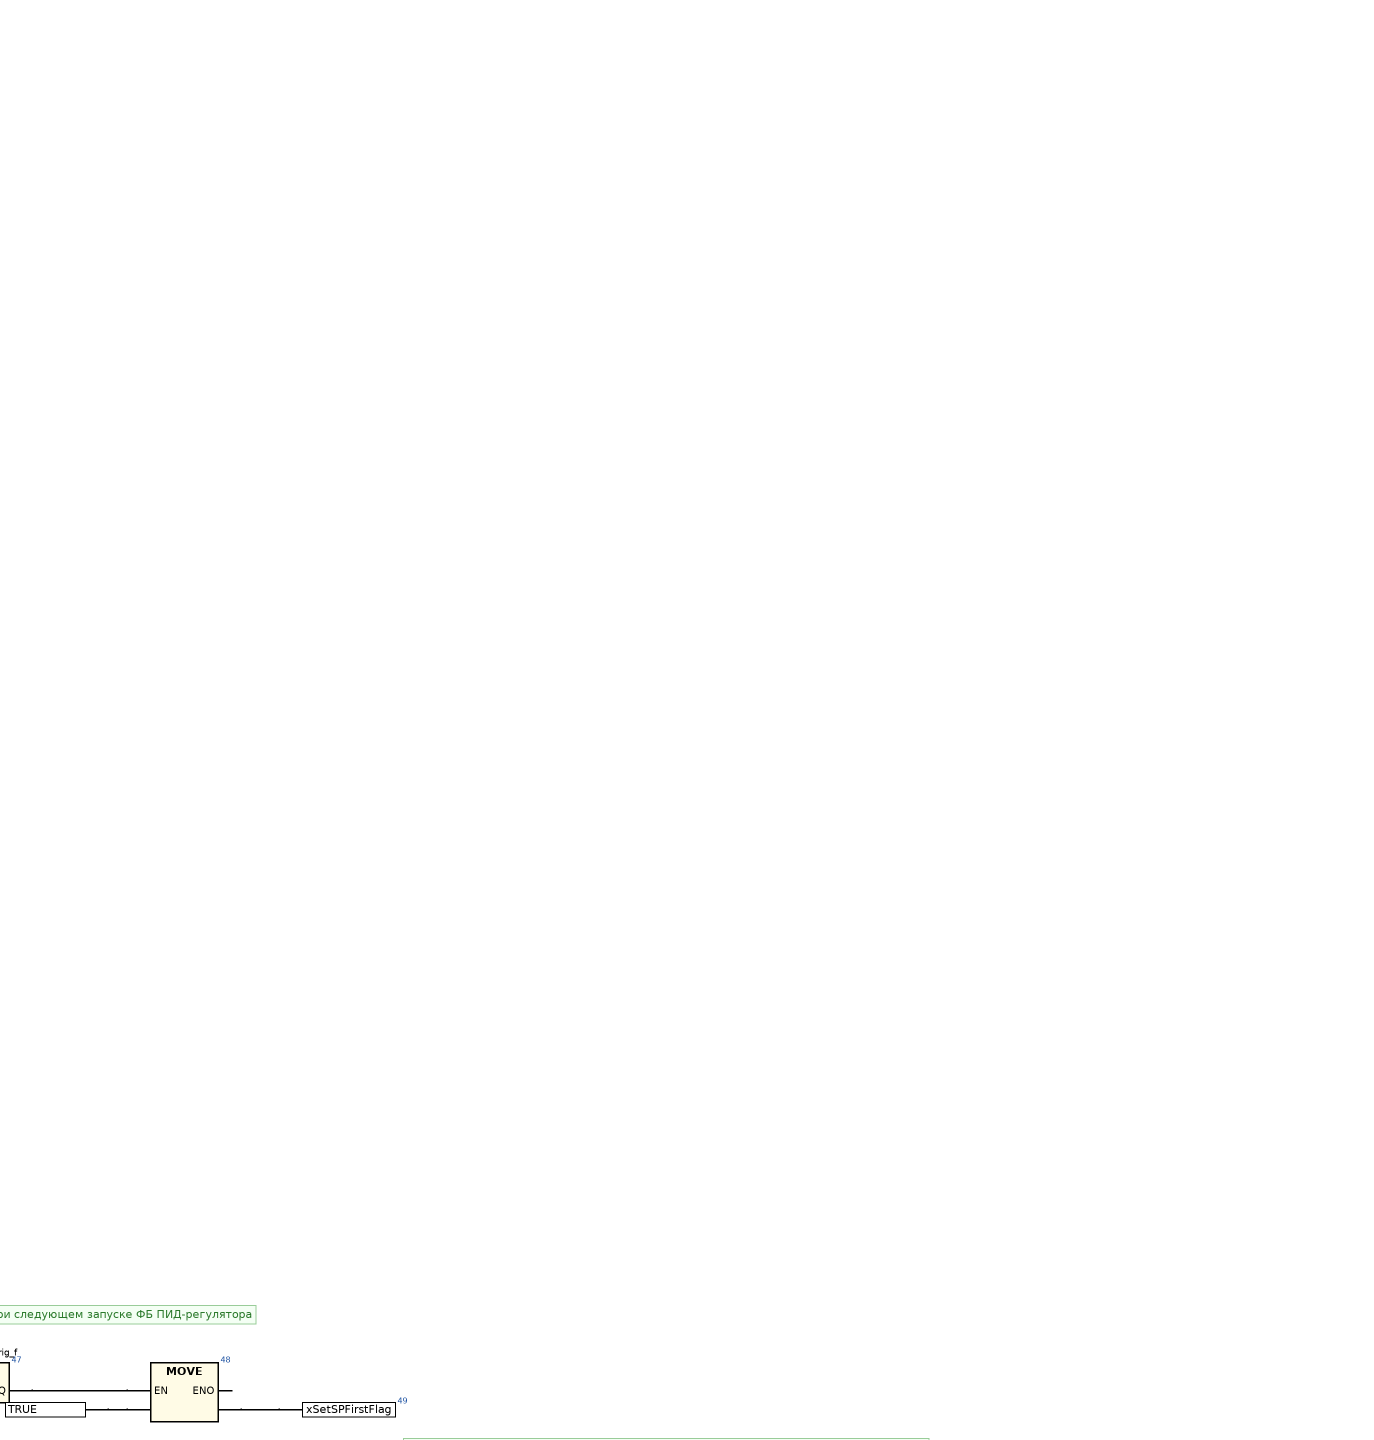
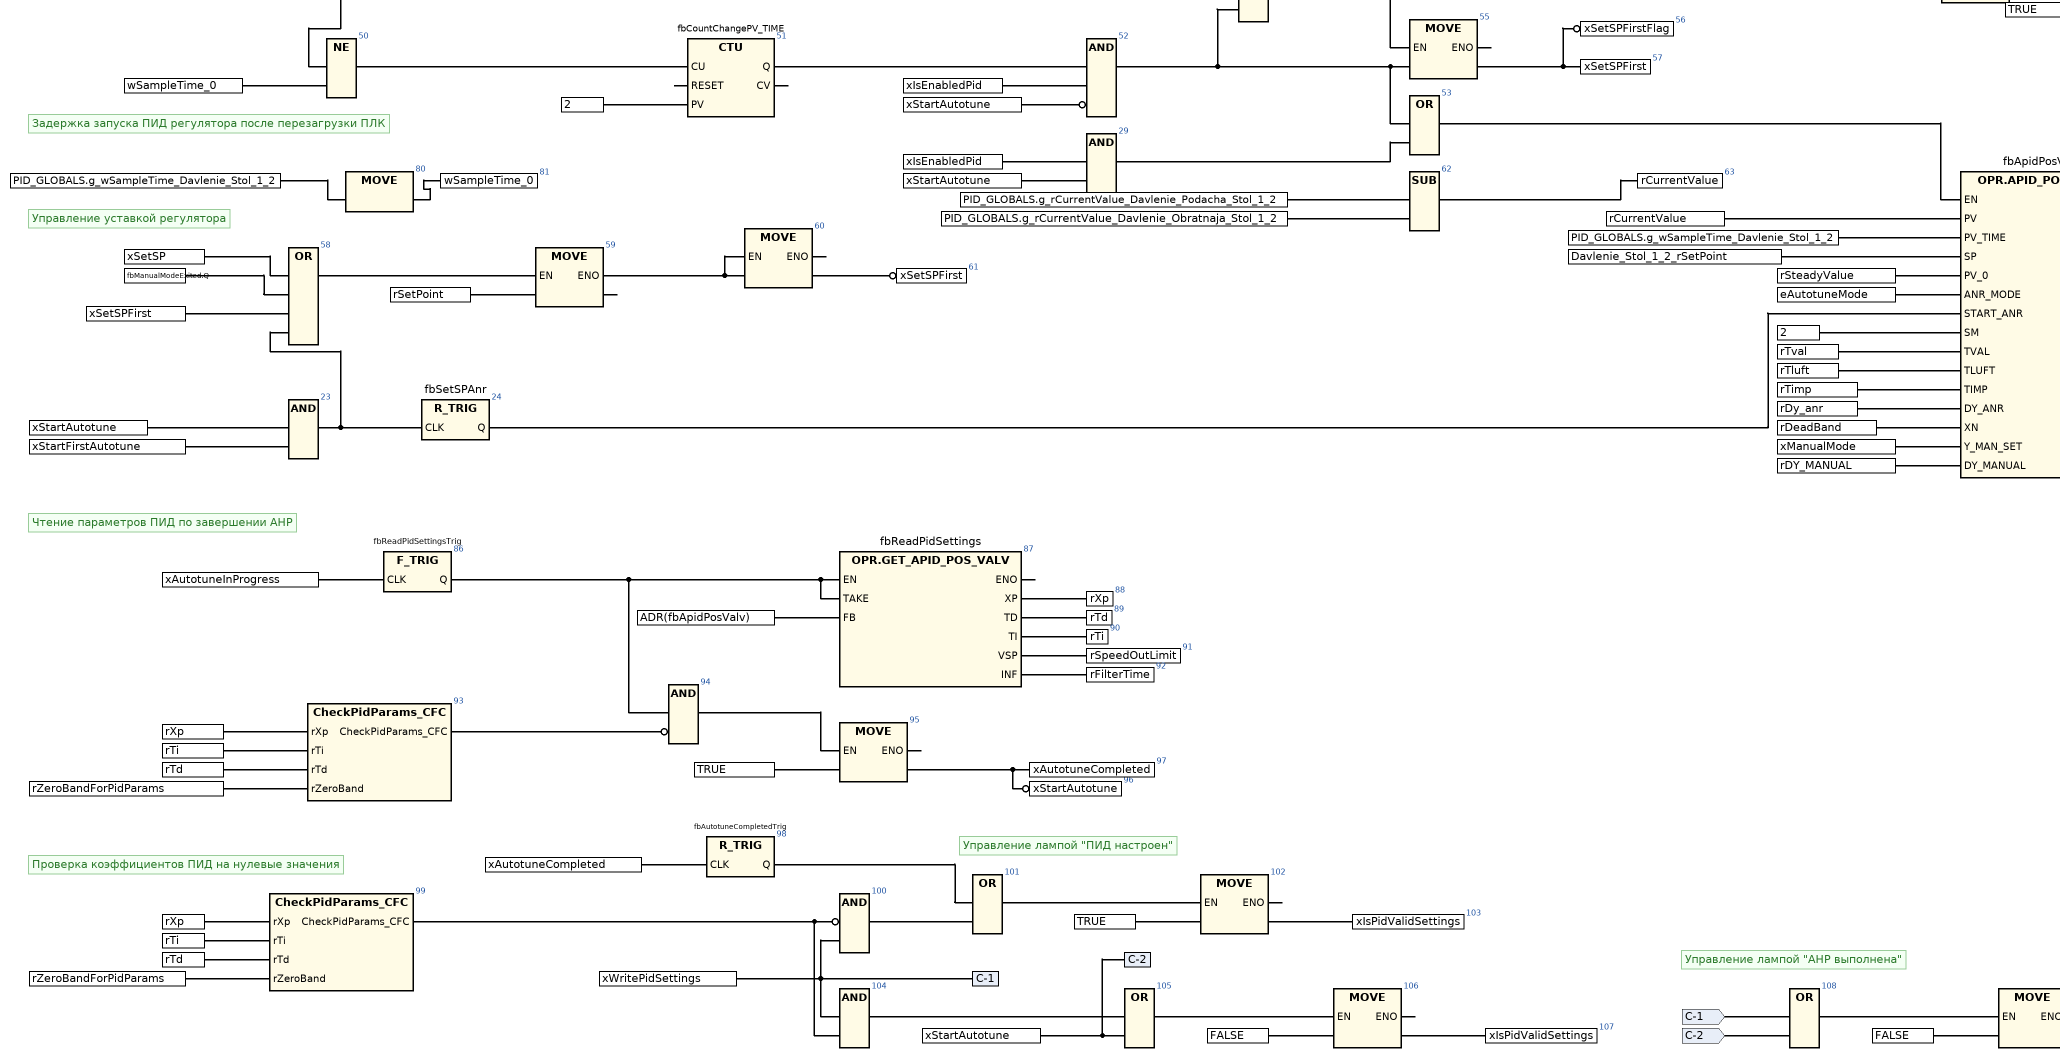
// Запись параметров ПИД при запуске контроллера, в случае не нулевых коэффициентов
_w1 := CheckPidParams_CFC(rXp := rXp, rTi := rTi, rTd := rTd, rZeroBand := rZeroBandForPidParams);
fbWritePidSettingsTrig(CLK := xWritePidSettings); // R_TRIG
_w2 := xWritePidSettingsAfterReboot AND NOT _w1;
IF _w2 THEN _w3 := _w2; END_IF
xWritePidSettingsAfterReboot := NOT _w3;
fbWritePidSettingsAfterRebootTrig(CLK := _w3); // R_TRIG
fbWritePidSettings(
    SETUP := fbWritePidSettingsAfterRebootTrig.Q OR fbWritePidSettingsTrig.Q,
    XP := rXp,
    TD := rTd,
    TI := rTi,
    VSP := rSpeedOutLimit,
    INF := rFilterTime,
    FB := ADR(fbApidPosValv)); // OPR.SET_APID_POS_VALV
// Ручное управление
fbManualModeExited(CLK := xManualMode); // F_TRIG
// Запись параметров ПИД пользователем
IF fbManualModeExited.Q AND NOT xStartAutotune THEN _w4 := rCurrentValue; END_IF
// При установке ручного управления PV=>SP
rSetPoint := _w4;
// Выключение и сброса параметров ФБ ПИД , после перезагрузки ПЛК, в случае ранее активной АНР или ручного режима
_w5 := xFirstCycle AND xAutotuneInProgress;
fbDy_manualTrig_r(CLK := xManual_set); // R_TRIG
IF fbDy_manualTrig_r.Q THEN _w6 := rManual_mean; END_IF
// Запись команд ручного управления
rDY_MANUAL := _w6;
// Сброса параметров основного ФБ ПИД перед пуском АНР
fbReset(CLK := xReset); // R_TRIG
IF fbReset.Q THEN _w7 := fbApidPosValvReset; END_IF
fbApidPosValv := _w7;
fbDy_manualTrig_f(CLK := fbDy_manualTrig_r.Q); // F_TRIG
IF fbDy_manualTrig_f.Q THEN _w8 := REAL#0.0; END_IF
rDY_MANUAL := _w8;
IF xFirstCycle THEN _w9 := xFirstCycle; END_IF
_w10 := xStartAutotune AND xStartFirstAutotune;
fbSetSPAnr(CLK := _w10); // R_TRIG
// Остановка (перемещение задвижки в исходное положение) при активации ручного режима. Срабатывает только в случае, когда задвижка отрабатывает последнее воздействие от АНР
fbDy_manualTrig_r_anr(CLK := xManualMode AND xAutotuneInProgress); // R_TRIG
fbDy_manualTrig_f_anr(CLK := fbDy_manualTrig_r_anr.Q); // F_TRIG
_w11 := SEL(fbApidPosValv.MORE, 0, -1);
_w12 := xIsEnabledPid AND xStartAutotune;
fbOffReset(CLK := _w5 OR xFirstCycle AND xManualMode); // R_TRIG
IF fbOffReset.Q THEN _w13 := fbOffReset.Q; END_IF
xReset := _w13;
fbDy_manualTrig_f_anr_0(CLK := fbDy_manualTrig_f_anr.Q); // F_TRIG
IF fbDy_manualTrig_f_anr_0.Q THEN _w14 := REAL#0.0; END_IF
rDY_MANUAL := _w14;
xFirstCycle := NOT _w9;
_w15 := SEL(fbApidPosValv.LESS, 0, 1);
IF fbOffReset.Q THEN _w16 := FALSE; END_IF
xIsEnabledPid := _w16;
xManualMode := _w16;
IF fbDy_manualTrig_f_anr.Q THEN _w17 := (_w11 + _w15) * rDy_anr * 0.01; END_IF
rDY_MANUAL := _w17;
// Установка флага на запись уставки при следующем запуске ФБ ПИД-регулятора
fbEnabledPidTrig_f(CLK := xIsEnabledPid); // F_TRIG
IF fbEnabledPidTrig_f.Q THEN _w18 := TRUE; END_IF
xSetSPFirstFlag := _w18;
fbCountChangePV_TIME(CU := PID_GLOBALS.g_wSampleTime_Davlenie_Stol_1_2 <> wSampleTime_0, PV := 2); // CTU
_w19 := fbCountChangePV_TIME.Q AND xIsEnabledPid AND NOT xStartAutotune;
_w20 := _w19 OR _w12;
// Запись уставки, при первом пуске ФБ ПИД
IF xSetSPFirstFlag AND _w19 THEN _w21 := _w19; END_IF
xSetSPFirstFlag := NOT _w21;
xSetSPFirst := _w21;
// Управление уставкой регулятора
_w22 := xSetSP OR fbManualModeExited.Q OR xSetSPFirst OR _w10;
IF _w22 THEN (* rSetPoint; result not used *) END_IF
IF _w22 THEN _w23 := _w22; END_IF
xSetSPFirst := NOT _w23;
rCurrentValue := PID_GLOBALS.g_rCurrentValue_Davlenie_Podacha_Stol_1_2 - PID_GLOBALS.g_rCurrentValue_Davlenie_Obratnaja_Stol_1_2;
_w24 := _w20;
IF _w24 THEN
    fbApidPosValv(
        PV := rCurrentValue,
        PV_TIME := PID_GLOBALS.g_wSampleTime_Davlenie_Stol_1_2,
        SP := Davlenie_Stol_1_2_rSetPoint,
        PV_0 := rSteadyValue,
        ANR_MODE := eAutotuneMode,
        START_ANR := fbSetSPAnr.Q,
        SM := 2,
        TVAL := rTval,
        TLUFT := rTluft,
        TIMP := rTimp,
        DY_ANR := rDy_anr,
        XN := rDeadBand,
        Y_MAN_SET := xManualMode,
        DY_MANUAL := rDY_MANUAL); // OPR.APID_POS_VALV
END_IF
xStartFirstAutotune := _w24;
xMore := fbApidPosValv.LESS;
xLess := fbApidPosValv.MORE;
xAutotuneInProgress := fbApidPosValv.ANR_WORK;
ePidError := fbApidPosValv.ERROR;
ePidState := fbApidPosValv.STATE;
rYsm := 1 - fbApidPosValv.YSM;
xDendl := fbApidPosValv.DENDH;
xDendh := fbApidPosValv.DENDL;
rYsm_scale := fbApidPosValv.YSM * 100.0;
// Управление сигнальной лампой (Вкл. - ОК!), указывающей на отсутствие регулирования
xSetManualOK := NOT fbApidPosValv.LESS AND NOT fbApidPosValv.MORE OR xAutotuneInProgress;
// Задержка запуска ПИД регулятора после перезагрузки ПЛК
wSampleTime_0 := PID_GLOBALS.g_wSampleTime_Davlenie_Stol_1_2;
// Передача выходов ФБ ПИД глобальным переменным, управляющих задвижкой
PID_GLOBALS.xOut_More_Davlenie_Stol_1_2 := xMore;
PID_GLOBALS.xOut_Less_Davlenie_Stol_1_2 := xLess;
// Чтение параметров ПИД по завершении АНР
fbReadPidSettingsTrig(CLK := xAutotuneInProgress); // F_TRIG
IF fbReadPidSettingsTrig.Q THEN
    fbReadPidSettings(TAKE := fbReadPidSettingsTrig.Q, FB := ADR(fbApidPosValv)); // OPR.GET_APID_POS_VALV
END_IF
rXp := fbReadPidSettings.XP;
rTd := fbReadPidSettings.TD;
rTi := fbReadPidSettings.TI;
rSpeedOutLimit := fbReadPidSettings.VSP;
rFilterTime := fbReadPidSettings.INF;
_w25 := CheckPidParams_CFC(rXp := rXp, rTi := rTi, rTd := rTd, rZeroBand := rZeroBandForPidParams);
IF fbReadPidSettingsTrig.Q AND NOT _w25 THEN _w26 := TRUE; END_IF
xStartAutotune := NOT _w26;
xAutotuneCompleted := _w26;
fbAutotuneCompletedTrig(CLK := xAutotuneCompleted); // R_TRIG
// Проверка коэффициентов ПИД на нулевые значения
_w27 := CheckPidParams_CFC(rXp := rXp, rTi := rTi, rTd := rTd, rZeroBand := rZeroBandForPidParams);
// Управление лампой "ПИД настроен"
IF fbAutotuneCompletedTrig.Q OR NOT _w27 AND xWritePidSettings THEN _w28 := TRUE; END_IF
xIsPidValidSettings := _w28;
IF xWritePidSettings AND _w27 OR xStartAutotune THEN _w29 := FALSE; END_IF
xIsPidValidSettings := _w29;
// Управление лампой "АНР выполнена"
IF xWritePidSettings OR xStartAutotune THEN _w30 := FALSE; END_IF
xAutotuneCompleted := _w30;

END_PROGRAM

// Device/Application/CFC_Temperatura_PID/CheckPidParams_CFC
FUNCTION CheckPidParams_CFC : BOOL
VAR_INPUT
	rXp: 			REAL;						// Коэффициент передачи
	rTi:			REAL;						// Постоянная времени интегрирования
	rTd: 			REAL;						// Постоянная времени дифференцирования
	rZeroBand: 		REAL;						// Зона нулевых коэффициентов ПИД
END_VAR
VAR
	fbLimitAlarm:	MATH.LimitAlarm_LREAL;		// Проверка поподания значения коэффициента в указаную зону
	xXpInLimits: 	BOOL;						// Xp в зоне нулевых коэффициентов ПИД - TRUE
	xTdInLimits: 	BOOL;						// Td в зоне нулевых коэффициентов ПИД - TRUE
	xTiInLimits:	BOOL;						// Ti в зоне нулевых коэффициентов ПИД - TRUE
END_VAR

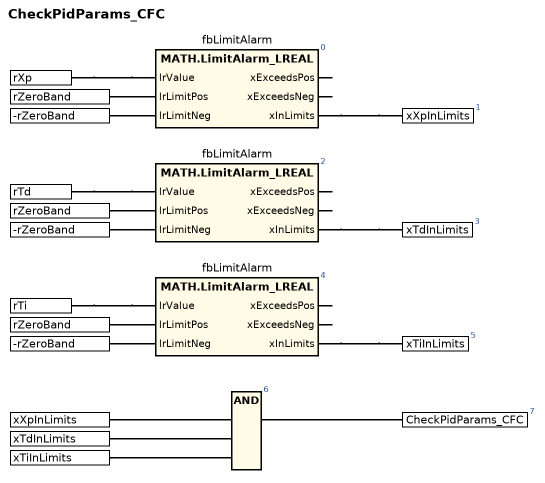
fbLimitAlarm(lrValue := rXp, lrLimitPos := rZeroBand, lrLimitNeg := -rZeroBand); // MATH.LimitAlarm_LREAL
xXpInLimits := fbLimitAlarm.xInLimits;
fbLimitAlarm(lrValue := rTd, lrLimitPos := rZeroBand, lrLimitNeg := -rZeroBand); // MATH.LimitAlarm_LREAL
xTdInLimits := fbLimitAlarm.xInLimits;
fbLimitAlarm(lrValue := rTi, lrLimitPos := rZeroBand, lrLimitNeg := -rZeroBand); // MATH.LimitAlarm_LREAL
xTiInLimits := fbLimitAlarm.xInLimits;
CheckPidParams_CFC := xXpInLimits AND xTdInLimits AND xTiInLimits;

END_FUNCTION

// Device/Application/CFC_Davlenie_PID/PLC_PRG_CFC_Davlenie_Stol_3_4
PROGRAM PLC_PRG_CFC_Davlenie_Stol_3_4
VAR
	(* входы регулятора *)
	//
	fbApidPosValv: 							OPR.APID_POS_VALV;		// ФБ ПИД регулятора с АНР
	fbDy_manualTrig_r:						R_TRIG;					// Детектор нажатия кнопки записи мощности в ручном режиме на вход DY_MANUAL
	fbDy_manualTrig_f:						F_TRIG;					// Детектор отпускания кнопки для сброса входа DY_MANUAL в 0
	rCurrentValue: 							REAL;					// Измеренное значение регулируемой величины
	rDY_MANUAL: 							REAL;					// Мощность, передаваемая на вход DY_MANUAL
	wSampleTime_0:							WORD;					// Значение PV_TIME в предыдущем цикле ПЛК
	fbCountChangePV_TIME: 					CTU;					// Счетчик циклов ПЛК, в которых происходило изменение PV_TIME
	xSetSP: 								BOOL;					// Команда на запись SP
	xSetSPFirst: 							BOOL;					// Команда на запись SP при запуске контроллера
	xSetSPFirstFlag: 						BOOL	:=	TRUE;		// Флаг записи SP при запуске контроллера
	fbEnabledPidTrig_f: 					F_TRIG;					// Детектор импульса на запись уставки в первом цикле ПЛК
	(* выходы регулятора *)
	//
	ePidState: 								OPR.STATE_PID;			// Состояние регулятора
	ePidError: 								OPR.ERROR_PID;			// Код ошибки регулятора
	xLess: 									BOOL;					// Сигнал на закрытие ИМ
	xMore:									BOOL;					// Сигнал на открытие ИМ
	rYsm: 									REAL;					// Расчетное положение выхода задвижки (для аналогового управления)
	rYsm_scale: 							REAL;					// Расчетное положение выхода задвижки, отображаемое на тренде
	xDendh:									BOOL;					// Признак достижения задвижкой 100%
	xDendl:									BOOL;					// Признак достижения задвижкой 0%
	(* параметры АНР *)
	//
	eAutotuneMode: 							OPR.TYPE_ANR;			// Тип автонастройки  (DYNAMIC - быстрый переход на новую уставку, но возможно перерегулирование; STABILITY - медленный переход на новую уставку, но с меньшим перерегулирование)
	xStartAutotune:							BOOL;					// Команда запуска АНР
	xStartFirstAutotune:					BOOL;					// Команда автоматического запуска АНР при включении контроллера (при нулевых параметрах ПИД)
	fbAutotuneCompletedTrig:				R_TRIG;					// Детектор импульса завершения АНР
	fbSetSPAnr: 							R_TRIG;					// Детектор импульса на запись SP при запуске АНР
	(* параметры ручного управления *)
	//
	fbManualModeExited: 					F_TRIG;					// Детектор импульса выхода из режима ручного управления
	xManual_set:							BOOL;					// Команда записи мощности в ручном режиме
	rManual_mean: 							REAL;					// Значение передаваемой мощности в ручном режиме
	xSetManualOK:							BOOL;					// Сигнал, указывающий на возможность безударного включения ручного режима (сигнал отсутствия регулирования)
	fbDy_manualTrig_r_anr: 					R_TRIG;					// Детектор импульса включения ручного режима при активной АНР
	fbDy_manualTrig_f_anr: 					F_TRIG;					// Задержка на цикл ПЛК на передачу параметра на вход rDy_anr
	fbDy_manualTrig_f_anr_0: 				F_TRIG;					// Сброс входа rDy_anr
	(* запись параметров регулятора *)
	//	
	xWritePidSettingsAfterReboot: 			BOOL	:=	TRUE;		// Команда восстановления параметров ПИД после перезагрузки контроллера
	xWritePidSettings:						BOOL;					// Команда записи параметров ПИД, введенных пользователем
	fbWritePidSettingsTrig: 				R_TRIG;					// Детектор импульса записи параметров ПИД пользователем
	(* ФБ записи параметров *)
	//
	fbWritePidSettings: 					OPR.SET_APID_POS_VALV;	// ФБ записи параметров ПИД
	fbWritePidSettingsAfterRebootTrig:		R_TRIG;					// Детектор импульса записи параметров ПИД после перезагрузки контроллера
	(* ФБ чтения параметров *)
	//	
	fbReadPidSettings: 						OPR.GET_APID_POS_VALV;	// ФБ чтения параметров ПИД
	fbReadPidSettingsTrig: 					F_TRIG;					// Детектор импульса чтения параметров ПИД
	(* Параметры выходов ПЛК *)
	//
	(*Параметры сброса ФБ ПИД*)
	fbApidPosValvReset: 					OPR.APID_POS_VALV;		// ФБ ПИД регулятора, используемый для сброса параметров основного ФБ ПИД перед запуском АНР
	xReset: 								BOOL;					// Команда на сброс ФБ ПИД
	fbReset: 								R_TRIG;					// Детектор импульса от переменной xReset
	xFirstCycle:						 	BOOL	:=	TRUE;		// Команда на сброс ФБ ПИД после перезагрузки ПЛК, в случае ранее активной АНР или ручного режима
	fbOffReset: 							R_TRIG;					// Детектор импульса от переменной xFirstCucle
	
	
	

END_VAR
VAR RETAIN
	Davlenie_Stol_3_4_rSetPoint: 			REAL; 					// Дельта давления
	xIsEnabledPid:							BOOL 	:= 	TRUE; 		// Состояние регулятора (TRUE - включен)
	rTval: 									REAL	:=	120;		// Время полного хода ИМ, сек
	rTluft:									REAL	:=	0.0;		// Время выборки люфта ИМ, сек
	rTimp:									REAL	:=	5;			// Минимальная длительность импульса, сек
	rDy_anr: 								REAL	:=	50.0;		// Размах мощности,%
	rSetPoint: 								REAL	:=	0.35;		// Уставка регулятора
	rSteadyValue: 							REAL	:=	0.3;		// Значение регулируемого параметра при нулевой мощности управляющего сигнала 
	rDeadBand: 								REAL 	:=	0.03;		// Зона нечувствительности ПИД
	rZeroBandForPidParams:					REAL	:=	0.001;		// Зона нулевых коэффициентов ПИД
	//
	rXp: 									REAL:=3.00;					// Полоса пропускания (100/Кр)
	rTi: 									REAL:=8.30;					// Постоянная времени интегрирования
	rTd: 									REAL:=1.53;					// Постоянная времени дифференцирования
	rSpeedOutLimit: 						REAL;					// Допустимая скорость изменения внутренней уставки ПИД
	rFilterTime: 							REAL;					// Постоянная времени входного фильтра ПИД
	//										
	xAutotuneCompleted:						BOOL;					// Импульс завершения АНР
	xIsPidValidSettings: 					BOOL;					// Сигнал настройки ПИД
	xManualMode: 							BOOL;					// Сигнал перевода ПИД в режим ручного управления
	xAutotuneInProgress:					BOOL;					// Флаг "Выполняется АНР"
END_VAR
VAR // added by the converter: edge detectors and wires of the graphical bodies
    _w1, _w8, _w11, _w13, _w14, _w15, _w25, _w27 : ANY;
    _w2, _w3, _w5, _w9, _w10, _w12, _w16, _w18, _w19, _w20, _w21, _w22, _w23, _w24, _w26, _w28, _w29, _w30 : BOOL;
    _w4, _w6, _w17 : REAL;
    _w7 : OPR.APID_POS_VALV;
END_VAR

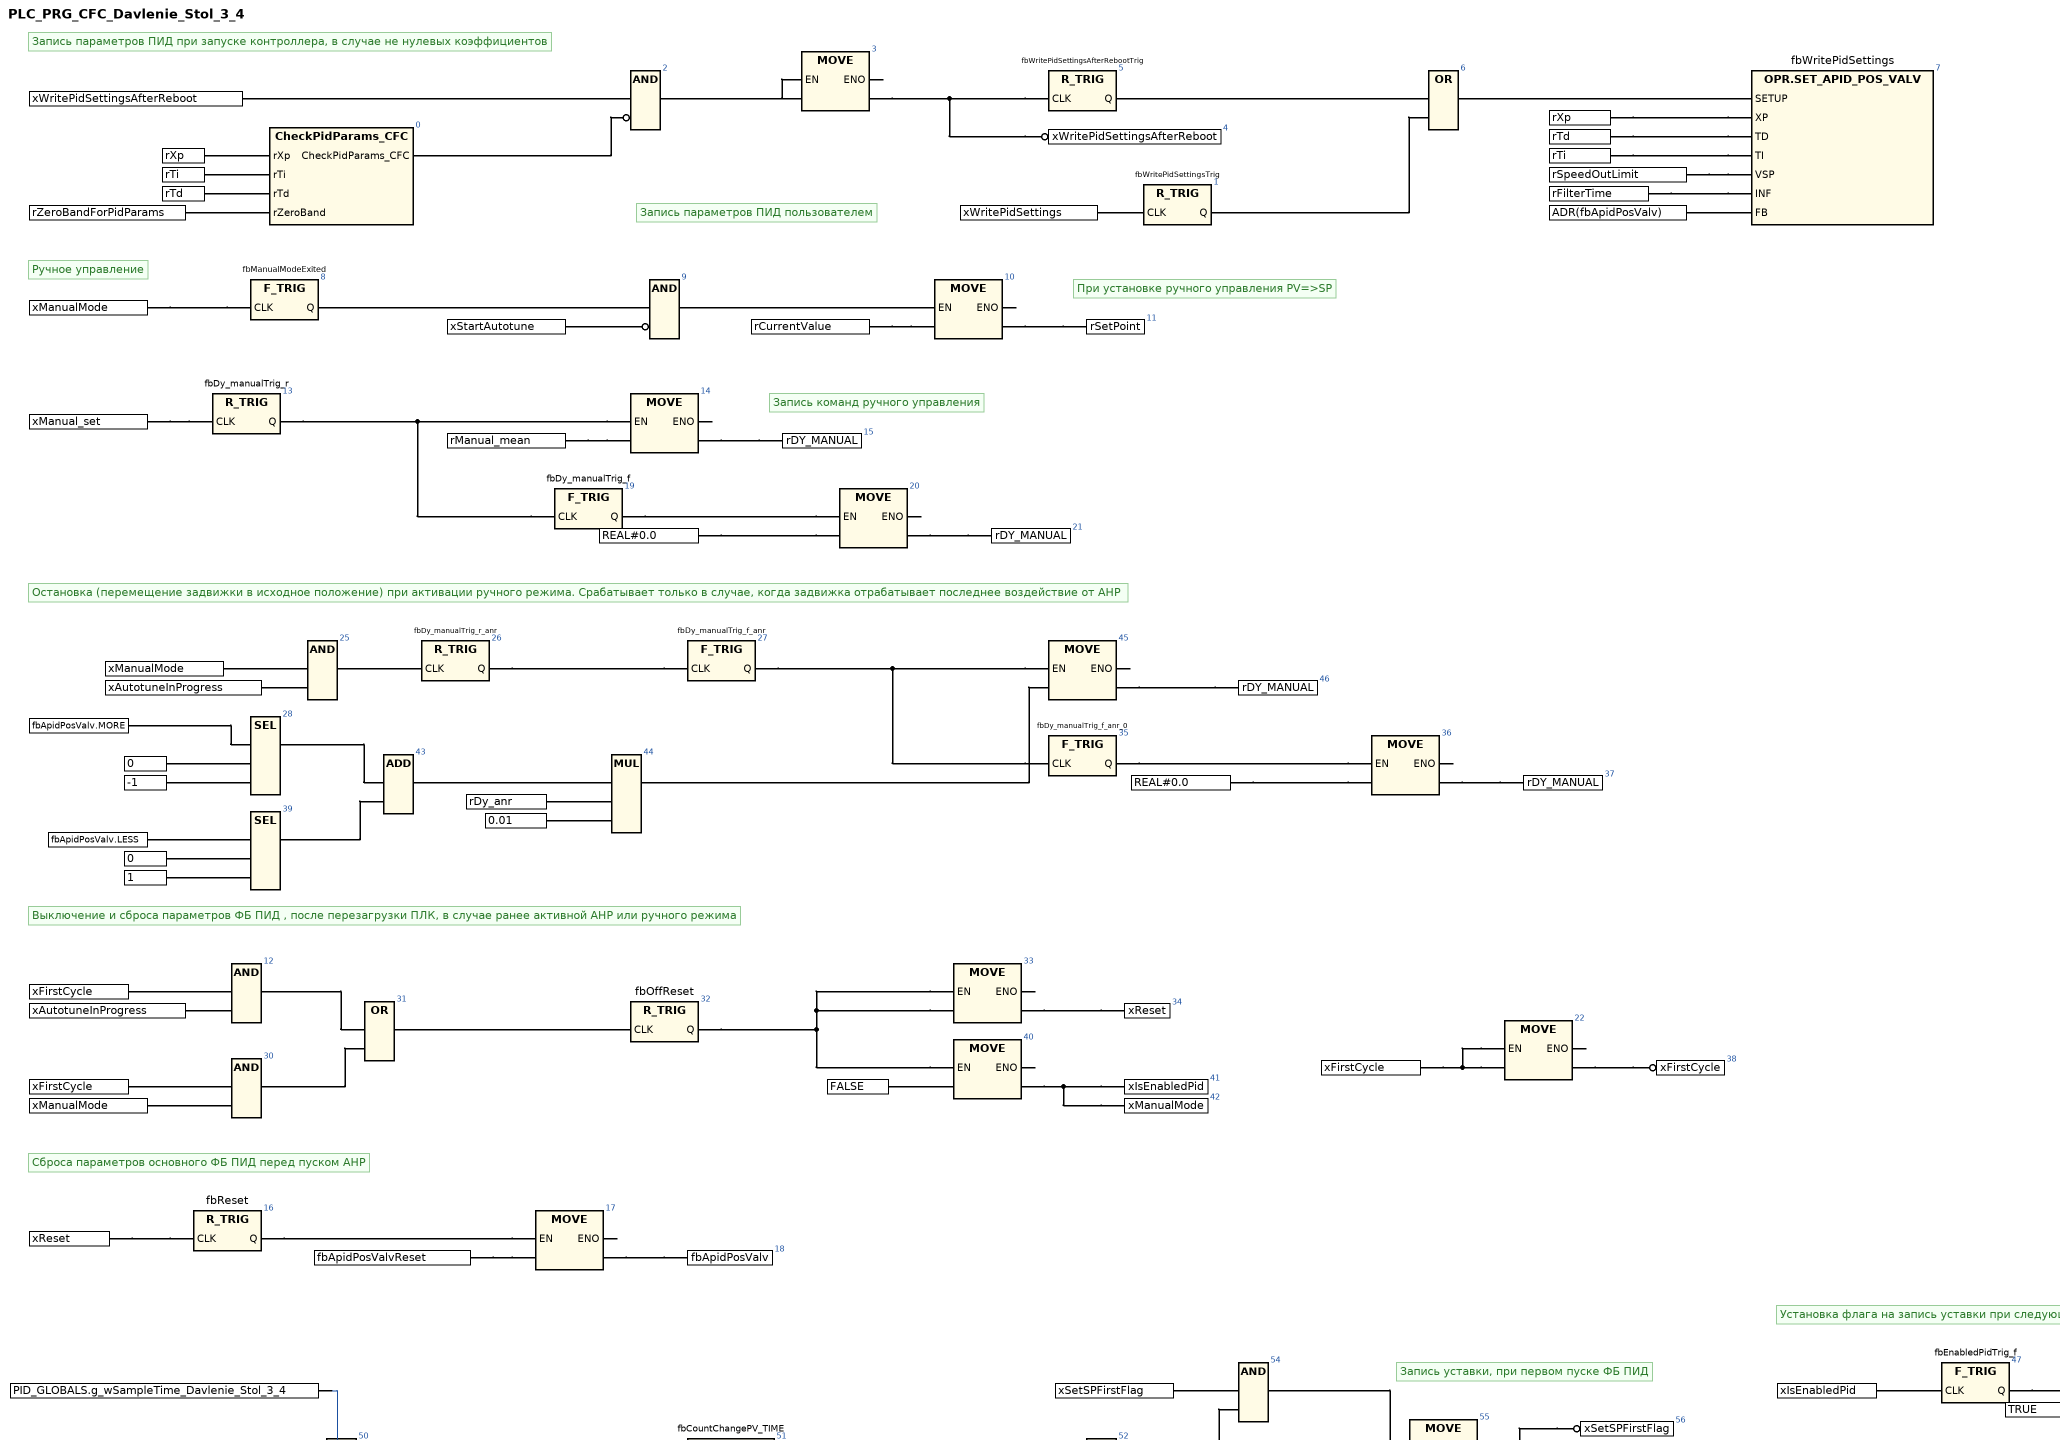
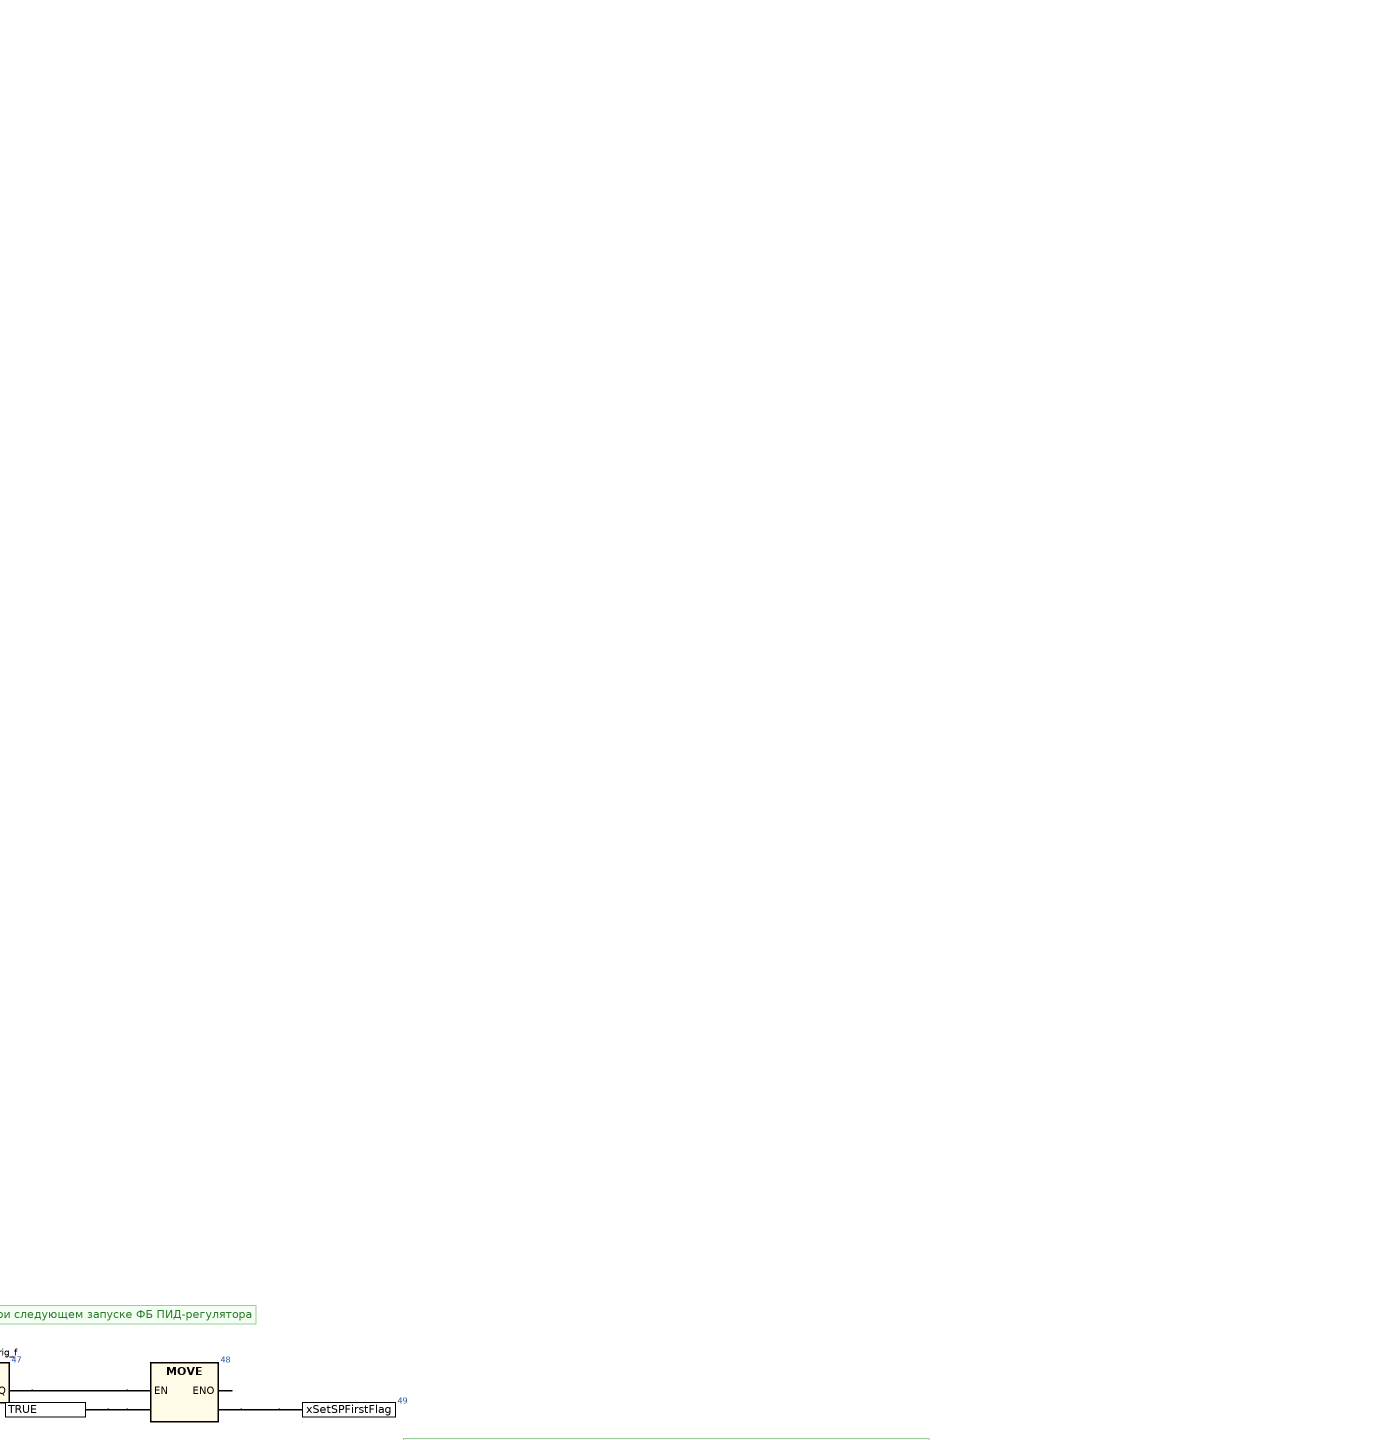
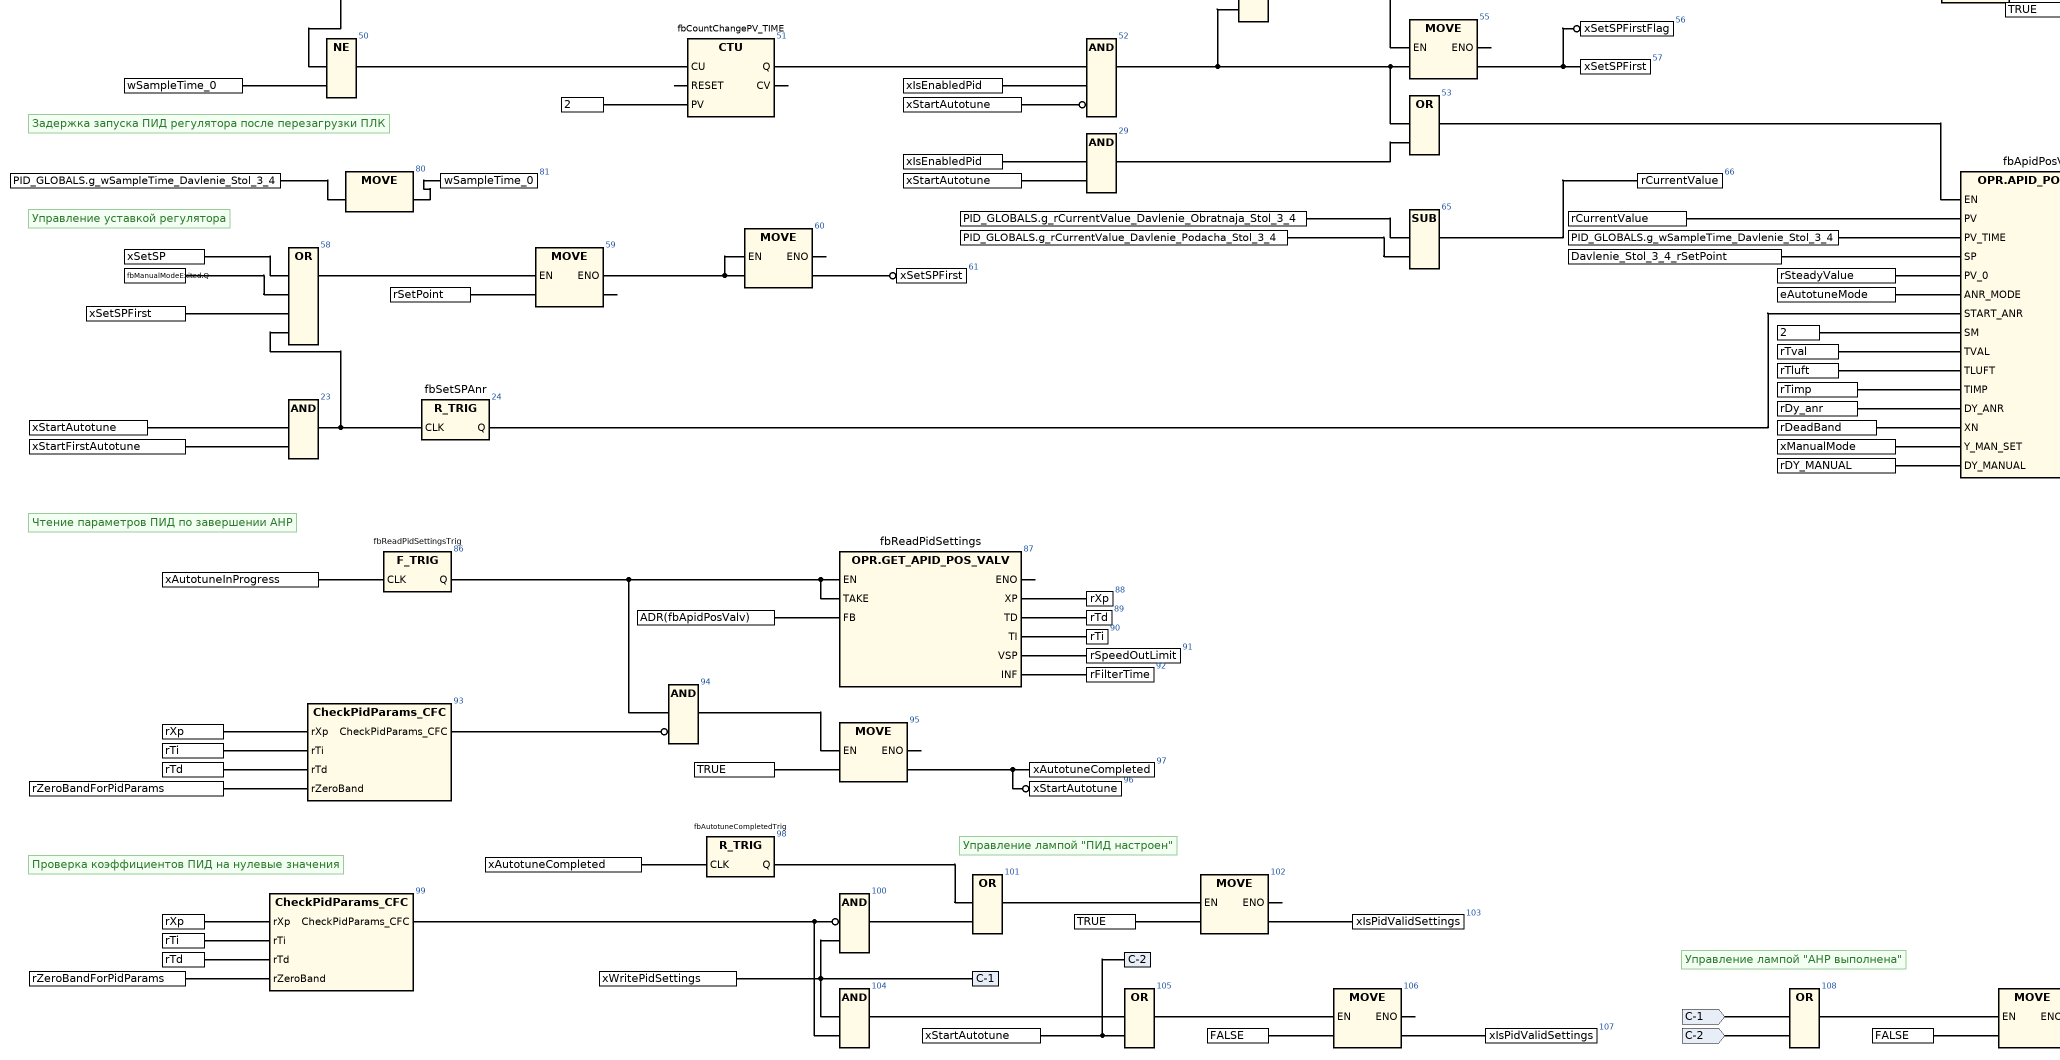
// Запись параметров ПИД при запуске контроллера, в случае не нулевых коэффициентов
_w1 := CheckPidParams_CFC(rXp := rXp, rTi := rTi, rTd := rTd, rZeroBand := rZeroBandForPidParams);
fbWritePidSettingsTrig(CLK := xWritePidSettings); // R_TRIG
_w2 := xWritePidSettingsAfterReboot AND NOT _w1;
IF _w2 THEN _w3 := _w2; END_IF
xWritePidSettingsAfterReboot := NOT _w3;
fbWritePidSettingsAfterRebootTrig(CLK := _w3); // R_TRIG
fbWritePidSettings(
    SETUP := fbWritePidSettingsAfterRebootTrig.Q OR fbWritePidSettingsTrig.Q,
    XP := rXp,
    TD := rTd,
    TI := rTi,
    VSP := rSpeedOutLimit,
    INF := rFilterTime,
    FB := ADR(fbApidPosValv)); // OPR.SET_APID_POS_VALV
// Ручное управление
fbManualModeExited(CLK := xManualMode); // F_TRIG
// Запись параметров ПИД пользователем
IF fbManualModeExited.Q AND NOT xStartAutotune THEN _w4 := rCurrentValue; END_IF
// При установке ручного управления PV=>SP
rSetPoint := _w4;
// Выключение и сброса параметров ФБ ПИД , после перезагрузки ПЛК, в случае ранее активной АНР или ручного режима
_w5 := xFirstCycle AND xAutotuneInProgress;
fbDy_manualTrig_r(CLK := xManual_set); // R_TRIG
IF fbDy_manualTrig_r.Q THEN _w6 := rManual_mean; END_IF
// Запись команд ручного управления
rDY_MANUAL := _w6;
// Сброса параметров основного ФБ ПИД перед пуском АНР
fbReset(CLK := xReset); // R_TRIG
IF fbReset.Q THEN _w7 := fbApidPosValvReset; END_IF
fbApidPosValv := _w7;
fbDy_manualTrig_f(CLK := fbDy_manualTrig_r.Q); // F_TRIG
IF fbDy_manualTrig_f.Q THEN _w8 := REAL#0.0; END_IF
rDY_MANUAL := _w8;
IF xFirstCycle THEN _w9 := xFirstCycle; END_IF
_w10 := xStartAutotune AND xStartFirstAutotune;
fbSetSPAnr(CLK := _w10); // R_TRIG
// Остановка (перемещение задвижки в исходное положение) при активации ручного режима. Срабатывает только в случае, когда задвижка отрабатывает последнее воздействие от АНР
fbDy_manualTrig_r_anr(CLK := xManualMode AND xAutotuneInProgress); // R_TRIG
fbDy_manualTrig_f_anr(CLK := fbDy_manualTrig_r_anr.Q); // F_TRIG
_w11 := SEL(fbApidPosValv.MORE, 0, -1);
_w12 := xIsEnabledPid AND xStartAutotune;
fbOffReset(CLK := _w5 OR xFirstCycle AND xManualMode); // R_TRIG
IF fbOffReset.Q THEN _w13 := fbOffReset.Q; END_IF
xReset := _w13;
fbDy_manualTrig_f_anr_0(CLK := fbDy_manualTrig_f_anr.Q); // F_TRIG
IF fbDy_manualTrig_f_anr_0.Q THEN _w14 := REAL#0.0; END_IF
rDY_MANUAL := _w14;
xFirstCycle := NOT _w9;
_w15 := SEL(fbApidPosValv.LESS, 0, 1);
IF fbOffReset.Q THEN _w16 := FALSE; END_IF
xIsEnabledPid := _w16;
xManualMode := _w16;
IF fbDy_manualTrig_f_anr.Q THEN _w17 := (_w11 + _w15) * rDy_anr * 0.01; END_IF
rDY_MANUAL := _w17;
// Установка флага на запись уставки при следующем запуске ФБ ПИД-регулятора
fbEnabledPidTrig_f(CLK := xIsEnabledPid); // F_TRIG
IF fbEnabledPidTrig_f.Q THEN _w18 := TRUE; END_IF
xSetSPFirstFlag := _w18;
fbCountChangePV_TIME(CU := PID_GLOBALS.g_wSampleTime_Davlenie_Stol_3_4 <> wSampleTime_0, PV := 2); // CTU
_w19 := fbCountChangePV_TIME.Q AND xIsEnabledPid AND NOT xStartAutotune;
_w20 := _w19 OR _w12;
// Запись уставки, при первом пуске ФБ ПИД
IF xSetSPFirstFlag AND _w19 THEN _w21 := _w19; END_IF
xSetSPFirstFlag := NOT _w21;
xSetSPFirst := _w21;
// Управление уставкой регулятора
_w22 := xSetSP OR fbManualModeExited.Q OR xSetSPFirst OR _w10;
IF _w22 THEN (* rSetPoint; result not used *) END_IF
IF _w22 THEN _w23 := _w22; END_IF
xSetSPFirst := NOT _w23;
_w24 := _w20;
IF _w24 THEN
    fbApidPosValv(
        PV := rCurrentValue,
        PV_TIME := PID_GLOBALS.g_wSampleTime_Davlenie_Stol_3_4,
        SP := Davlenie_Stol_3_4_rSetPoint,
        PV_0 := rSteadyValue,
        ANR_MODE := eAutotuneMode,
        START_ANR := fbSetSPAnr.Q,
        SM := 2,
        TVAL := rTval,
        TLUFT := rTluft,
        TIMP := rTimp,
        DY_ANR := rDy_anr,
        XN := rDeadBand,
        Y_MAN_SET := xManualMode,
        DY_MANUAL := rDY_MANUAL); // OPR.APID_POS_VALV
END_IF
xStartFirstAutotune := _w24;
rCurrentValue := PID_GLOBALS.g_rCurrentValue_Davlenie_Obratnaja_Stol_3_4 - PID_GLOBALS.g_rCurrentValue_Davlenie_Podacha_Stol_3_4;
xMore := fbApidPosValv.LESS;
xLess := fbApidPosValv.MORE;
xAutotuneInProgress := fbApidPosValv.ANR_WORK;
ePidError := fbApidPosValv.ERROR;
ePidState := fbApidPosValv.STATE;
rYsm := 1 - fbApidPosValv.YSM;
xDendl := fbApidPosValv.DENDH;
xDendh := fbApidPosValv.DENDL;
rYsm_scale := fbApidPosValv.YSM * 100.0;
// Управление сигнальной лампой (Вкл. - ОК!), указывающей на отсутствие регулирования
xSetManualOK := NOT fbApidPosValv.LESS AND NOT fbApidPosValv.MORE OR xAutotuneInProgress;
// Задержка запуска ПИД регулятора после перезагрузки ПЛК
wSampleTime_0 := PID_GLOBALS.g_wSampleTime_Davlenie_Stol_3_4;
// Передача выходов ФБ ПИД глобальным переменным, управляющих задвижкой
PID_GLOBALS.xOut_More_Davlenie_Stol_3_4 := xMore;
PID_GLOBALS.xOut_Less_Davlenie_Stol_3_4 := xLess;
// Чтение параметров ПИД по завершении АНР
fbReadPidSettingsTrig(CLK := xAutotuneInProgress); // F_TRIG
IF fbReadPidSettingsTrig.Q THEN
    fbReadPidSettings(TAKE := fbReadPidSettingsTrig.Q, FB := ADR(fbApidPosValv)); // OPR.GET_APID_POS_VALV
END_IF
rXp := fbReadPidSettings.XP;
rTd := fbReadPidSettings.TD;
rTi := fbReadPidSettings.TI;
rSpeedOutLimit := fbReadPidSettings.VSP;
rFilterTime := fbReadPidSettings.INF;
_w25 := CheckPidParams_CFC(rXp := rXp, rTi := rTi, rTd := rTd, rZeroBand := rZeroBandForPidParams);
IF fbReadPidSettingsTrig.Q AND NOT _w25 THEN _w26 := TRUE; END_IF
xStartAutotune := NOT _w26;
xAutotuneCompleted := _w26;
fbAutotuneCompletedTrig(CLK := xAutotuneCompleted); // R_TRIG
// Проверка коэффициентов ПИД на нулевые значения
_w27 := CheckPidParams_CFC(rXp := rXp, rTi := rTi, rTd := rTd, rZeroBand := rZeroBandForPidParams);
// Управление лампой "ПИД настроен"
IF fbAutotuneCompletedTrig.Q OR NOT _w27 AND xWritePidSettings THEN _w28 := TRUE; END_IF
xIsPidValidSettings := _w28;
IF xWritePidSettings AND _w27 OR xStartAutotune THEN _w29 := FALSE; END_IF
xIsPidValidSettings := _w29;
// Управление лампой "АНР выполнена"
IF xWritePidSettings OR xStartAutotune THEN _w30 := FALSE; END_IF
xAutotuneCompleted := _w30;

END_PROGRAM

// Device/Application/CFC_Temperatura_PID/PLC_PRG_CFC_Temperatura_Stol_1
PROGRAM PLC_PRG_CFC_Temperatura_Stol_1
VAR
	ACTUATOR_3P_1:		OSCAT_BUILDING.ACTUATOR_3P;
	PID_1: 				PID;						// ФБ ПИД
	arx: 				BOOL;
	xMore:				BOOL;						// Сигнал открытия
	xLess: 				BOOL;						// Сигнал на закрытие
	
	TEST: 				BOOL;						// Переменная запускающая тестирование ФБ ACTUATOR_3P
	Pos: 				BYTE;						// Переменная принимающая позицию 3-х ходового клапана виртуальную
	ARE: BOOL;
	END_POS: BOOL;
	ERR: BOOL;
	STATUS: BYTE;
	F_TRIG_11: F_TRIG;
	TOF11: TOF;
END_VAR

VAR RETAIN	
	rXp: 									REAL:=1.5;					// Полоса пропускания (100/Кр)
	rTi: 									REAL:=25;					// Постоянная времени интегрирования
	rTd: 									REAL:=0.02;					// Постоянная времени дифференцирования
	Time_RUN:								TIME:=T#60S;				// Время хода 3-х ходового клапана
END_VAR

